METHOD Init : ITcoTaskStatus
VAR_INPUT
END_VAR
_closeTask.Restore();
Init := _closeTask.Invoke();
END_METHOD

PROPERTY InitTask : TcoCore.ITcoTask
GET
InitTask := _InitTask;
END_GET
END_PROPERTY

METHOD Open : ITcoTaskStatus
VAR_INPUT
END_VAR
_openTask.Restore();
Open := _openTask.Invoke();
END_METHOD

PROPERTY OpenTask : TcoCore.ITcoTask
GET
OpenTask := _OpenTask;
END_GET
END_PROPERTY

{warning 'Methodenimplementierung hinzufügen'}
METHOD Restore : TcoCore.ITcoRestorable
END_METHOD

{warning 'Methodenimplementierung hinzufügen'}
(*~
	<docu>
		<summary>
		    Custom service (manual, maintenance) logic.
			This method must be implemented in derived class.
		</summary>			
	</docu>	
~*)
METHOD PROTECTED ServiceMode
END_METHOD

PROPERTY Status : REFERENCE TO TcaSegmentDoorStatus
GET
Status REF= _status;
END_GET
END_PROPERTY

END_FUNCTION_BLOCK

// ---- Program/Handling/Dialogs/Handling_TeachRack_DlgContent.TcPOU
FUNCTION_BLOCK Handling_TeachRack_DlgContent EXTENDS TcoCore.TcoInputDialogContentContainer
VAR
	{attribute addProperty Name "<#Recipe#>"}
	Recipe:STRING;
	{attribute addProperty Name "<#Qantity#>"}
	RequiredQuantity:INT;
	{attribute addProperty Name "<#Timeout#>"}
	Timeout:DATE_AND_TIME;
	{attribute addProperty Name "<#Exclude#>"}
	Exclude:BOOL;
END_VAR

PROPERTY Context : TcoCore.ITcoContext
GET
END_GET
END_PROPERTY

PROPERTY Identity : ULINT
GET
END_GET
END_PROPERTY

END_FUNCTION_BLOCK

// ---- Template/Component_Cylinder/Base/CylinderBase.TcPOU
FUNCTION_BLOCK ABSTRACT CylinderBase EXTENDS TcoCore.TcoComponent IMPLEMENTS ICylinder
VAR_INPUT
	(*~
		<docu>
			<summary>
				Home position sensor.
			</summary>	
		</docu>
	~*)
	{attribute addProperty Name "<#Home position sensor#>"}
	inAtHomePos : BOOL;
	(*~
		<docu>
			<summary>
				Working position sensor.
			</summary>	
		</docu>
	~*)
	{attribute addProperty Name "<#Work position sensor#>"}
	inAtWorkPos : BOOL;
END_VAR
VAR_OUTPUT
	(*~
		<docu>
			<summary>
				Move to working home position signal.
			</summary>	
		</docu>
	~*)
	{attribute addProperty Name "<#Move to home position actuator#>"}
	outToHomePos : BOOL;
	(*~
		<docu>
			<summary>
				Move to working posistion signal.
			</summary>	
		</docu>
	~*)
	{attribute addProperty Name "<#Move to work position actuator#>"}
	outToWorkPos : BOOL;
END_VAR

(*~
	<docu>
		<summary>
			Gets whether the piston is in home position. 		
		</summary>			
	</docu>	
~*)
PROPERTY AtHome : bool
GET
AtHome := THIS^.inAtHomePos;
END_GET
END_PROPERTY

(*~
	<docu>
		<summary>
			Gets whether the piston is in work position. 		
		</summary>			
	</docu>	
~*)
PROPERTY AtWork : bool
GET
AtWork := inAtWorkPos;
END_GET
END_PROPERTY

METHOD FB_init : BOOL
VAR_INPUT
	bInitRetains : BOOL; // if TRUE, the retain variables are initialized (warm start / cold start)
	bInCopyCode : BOOL;  // if TRUE, the instance afterwards gets moved into the copy code (online change)
	Parent : ITcoObject;
END_VAR
END_METHOD

(*~
	<docu>
		<summary>
			Gets the `MoveHomeTask` task that controls the moving of the cyclinder in home position.
			<remarks>			
				<note type="important">
					This is an abstract method and must be implemented in derived class.
				</note>
			</remarks>	 		
		</summary>			
	</docu>	
~*)
PROPERTY PUBLIC ABSTRACT MoveHomeTask : TcoCore.ITcoTask
GET
END_GET
END_PROPERTY

(*~
	<docu>
		<summary>
			Starts movement into home position. 		
		</summary>			
	</docu>	
~*)
METHOD MoveToHome : TcoCore.ITcoTaskStatus
MoveToHome := MoveHomeTask.Invoke();
END_METHOD

(*~
	<docu>
		<summary>
			Starts movement into work position. 		
		</summary>			
	</docu>	
~*)
METHOD MoveToWork :TcoCore.ITcoTaskStatus
MoveToWork := MoveWorkTask.Invoke();
END_METHOD

(*~
	<docu>
		<summary>
			Gets the `MoveWorkTask` task that controls the moving of the cyclinder into work position.
			<remarks>			
				<note type="important">
					This is an abstract method and must be implemented in derived class.
				</note>
			</remarks>	 		
		</summary>			
	</docu>	
~*)
PROPERTY PUBLIC ABSTRACT MoveWorkTask : TcoCore.ITcoTask
GET
END_GET
END_PROPERTY

(*~
	<docu>
		<summary>
			Restore all tasks of this instance into initial state.		 		 		
		</summary>			
	</docu>	
~*)
METHOD  Restore : ITcoRestorable
MoveHomeTask.Restore();
MoveWorkTask.Restore();
StopTask.Restore();
END_METHOD

METHOD PROTECTED  ServiceMode
END_METHOD

(*~
	<docu>
		<summary>
			Stops cyclinder movement.
		 	<remarks>			
				<note type="important">
					This method switched off the signals for the movement of the piston in both direction.
					However depending on the pnemumatics configuration the movement may contintue if designed in that way.
					THIS IS NOT A SAFETY FUCTION!
				</note>
			</remarks>	 		
		</summary>			
	</docu>	
~*)
METHOD Stop : TcoCore.ITcoTaskStatus
Stop := StopTask.Invoke();
END_METHOD

(*~
	<docu>
		<summary>
			Gets the `StopTask` task that controls the stopping cyclinder movement.
			<remarks>			
				<note type="important">
					This is an abstract method and must be implemented in derived class.
				</note>
			</remarks>	 		
		</summary>			
	</docu>	
~*)
PROPERTY PUBLIC ABSTRACT StopTask : TcoCore.ITcoTask
GET
END_GET
END_PROPERTY

END_FUNCTION_BLOCK

// ---- Template/Component_Cylinder/Base/TcoDoubleCylinderBase.TcPOU
FUNCTION_BLOCK ABSTRACT TcoDoubleCylinderBase EXTENDS TcoCore.TcoComponent IMPLEMENTS ITcoCylinder
VAR_IN_OUT
	(*~
		<docu>
			<summary>
				Home position sensor 1.
			</summary>	
		</docu>
	~*)
	{attribute addProperty Name "<#Home position sensor#> - 1"}
	inoAtHomePos1 : BOOL;
		(*~
		<docu>
			<summary>
				Home position sensor 2.
			</summary>	
		</docu>
	~*)
	{attribute addProperty Name "<#Home position sensor#> - 2"}
	inoAtHomePos2 : BOOL;
		(*~
		<docu>
			<summary>
				Working position sensor 1.
			</summary>	
		</docu>
	~*)
	{attribute addProperty Name "<#Work position sensor#> - 1"}
	inoAtWorkPos1 : BOOL;
	(*~
		<docu>
			<summary>
				Working position sensor 1.
			</summary>	
		</docu>
	~*)
	{attribute addProperty Name "<#Work position sensor#> - 2"}
	inoAtWorkPos2 : BOOL;
END_VAR
VAR_IN_OUT
	(*~
		<docu>
			<summary>
				Move to working home position signal.
			</summary>	
		</docu>
	~*)
	{attribute addProperty Name "<#Move to home position actuator#>"}
	inoToHomePos : BOOL;
	(*~
		<docu>
			<summary>
				Move to working posistion signal.
			</summary>	
		</docu>
	~*)
	{attribute addProperty Name "<#Move to work position actuator#>"}
	inoToWorkPos : BOOL;
END_VAR
VAR
	(*~
		<docu>
			<summary>
				Home position sensor.
			</summary>	
		</docu>
	~*)
	{attribute addProperty Name "<#Home position sensor#>"}
	_atHomePos : BOOL;
	(*~
		<docu>
			<summary>
				Working position sensor.
			</summary>	
		</docu>
	~*)
	{attribute addProperty Name "<#Work position sensor#>"}
	_atWorkPos : BOOL;
	(*~
		<docu>
			<summary>
				Move to working home position signal.
			</summary>	
		</docu>
	~*)
	{attribute addProperty Name "<#Move to home position actuator#>"}
	_toHomePos : BOOL;
	(*~
		<docu>
			<summary>
				Move to working posistion signal.
			</summary>	
		</docu>
	~*)
	{attribute addProperty Name "<#Move to work position actuator#>"}
	_toWorkPos : BOOL;
END_VAR

VAR
	{attribute addProperty Name "<#Home sensor signal 1#>"}
	_atHomePos1SignalInfo : TcoCore.TcoSignalInfo;
	{attribute addProperty Name "<#Home sensor signal 2#>"}
	_atHomePos2SignalInfo : TcoCore.TcoSignalInfo;
	{attribute addProperty Name "<#Work sensor signal 1#>"}
    _atWorkPos1SignalInfo : TcoCore.TcoSignalInfo;
	{attribute addProperty Name "<#Work sensor signal 2#>"}
    _atWorkPos2SignalInfo : TcoCore.TcoSignalInfo;
	{attribute addProperty Name "<#Move to home position signal#>"}
    _toHomePosSignalInfo : TcoCore.TcoSignalInfo;
	{attribute addProperty Name "<#Move to work position signal#>"}
    _toWorkPosSignalInfo : TcoCore.TcoSignalInfo;
END_VAR

IF(__ISVALIDREF(inoAtHomePos1) AND __ISVALIDREF(inoAtHomePos2)) THEN _atHomePos := inoAtHomePos1 AND inoAtHomePos2; _atHomePos1SignalInfo.GetSignalInfo(SIZEOF(inoAtHomePos1), ADR(inoAtHomePos1));_atHomePos2SignalInfo.GetSignalInfo(SIZEOF(inoAtHomePos2), ADR(inoAtHomePos2)); END_IF;
IF(__ISVALIDREF(inoAtWorkPos1) AND __ISVALIDREF(inoAtWorkPos2)) THEN _atWorkPos := inoAtWorkPos1 AND inoAtWorkPos2; _atWorkPos1SignalInfo.GetSignalInfo(SIZEOF(inoAtWorkPos1), ADR(inoAtWorkPos1));_atWorkPos2SignalInfo.GetSignalInfo(SIZEOF(inoAtWorkPos2), ADR(inoAtWorkPos2)); END_IF;
IF(__ISVALIDREF(inoToHomePos)) THEN inoToHomePos := _toHomePos; _toHomePosSignalInfo.GetSignalInfo(SIZEOF(inoToHomePos), ADR(inoToHomePos)); END_IF;
IF(__ISVALIDREF(inoToWorkPos)) THEN inoToWorkPos := _toWorkPos; _toWorkPosSignalInfo.GetSignalInfo(SIZEOF(inoToWorkPos), ADR(inoToWorkPos)); END_IF;

(*~
	<docu>
		<summary>
			Gets whether the piston is in home position. 		
		</summary>			
	</docu>	
~*)
PROPERTY AtHome : bool
GET
AtHome := THIS^._atHomePos;
END_GET
END_PROPERTY

(*~
	<docu>
		<summary>
			Gets whether the piston is in work position. 		
		</summary>			
	</docu>	
~*)
PROPERTY AtWork : bool
GET
AtWork := _atWorkPos;
END_GET
END_PROPERTY

METHOD FB_init : BOOL
VAR_INPUT
	bInitRetains : BOOL; // if TRUE, the retain variables are initialized (warm start / cold start)
	bInCopyCode : BOOL;  // if TRUE, the instance afterwards gets moved into the copy code (online change)
	ParentObject : ITcoObject;	
END_VAR
END_METHOD

(*~
	<docu>
		<summary>
			Gets the `MoveHomeTask` task that controls the moving of the cyclinder in home position.
			<remarks>			
				<note type="important">
					This is an abstract method and must be implemented in derived class.
				</note>
			</remarks>	 		
		</summary>			
	</docu>	
~*)
PROPERTY PUBLIC ABSTRACT MoveHomeTask : TcoCore.ITcoTask
GET
END_GET
END_PROPERTY

(*~
	<docu>
		<summary>
			Starts movement into home position. 		
		</summary>			
	</docu>	
~*)
METHOD MoveToHome : TcoCore.ITcoTaskStatus
IF(MoveHomeTask <> 0) THEN 
	MoveToHome := MoveHomeTask.Invoke();
END_IF;
END_METHOD

(*~
	<docu>
		<summary>
			Starts movement into work position. 		
		</summary>			
	</docu>	
~*)
METHOD MoveToWork :TcoCore.ITcoTaskStatus
IF(MoveWorkTask <> 0) THEN
	MoveToWork := MoveWorkTask.Invoke();
END_IF;
END_METHOD

(*~
	<docu>
		<summary>
			Gets the `MoveWorkTask` task that controls the moving of the cyclinder into work position.
			<remarks>			
				<note type="important">
					This is an abstract method and must be implemented in derived class.
				</note>
			</remarks>	 		
		</summary>			
	</docu>	
~*)
PROPERTY PUBLIC ABSTRACT MoveWorkTask : TcoCore.ITcoTask
GET
END_GET
END_PROPERTY

(*~
	<docu>
		<summary>
			Restore all tasks of this instance into initial state.		 		 		
		</summary>			
	</docu>	
~*)
METHOD  Restore : ITcoRestorable
IF(MoveHomeTask <> 0) THEN MoveHomeTask.Restore(); END_IF;
IF(MoveWorkTask <> 0) THEN MoveWorkTask.Restore(); END_IF;
IF(StopTask <> 0) THEN StopTask.Restore(); END_IF;
END_METHOD

METHOD PROTECTED  ServiceMode
END_METHOD

(*~
	<docu>
		<summary>
			Stops cyclinder movement.
		 	<remarks>			
				<note type="important">
					This method switched off the signals for the movement of the piston in both direction.
					However depending on the pnemumatics configuration the movement may contintue if designed in that way.
					THIS IS NOT A SAFETY FUCTION!
				</note>
			</remarks>	 		
		</summary>			
	</docu>	
~*)
METHOD Stop : TcoCore.ITcoTaskStatus
IF(StopTask <> 0) THEN
	Stop := StopTask.Invoke();
END_IF;
END_METHOD

(*~
	<docu>
		<summary>
			Gets the `StopTask` task that controls the stopping cyclinder movement.
			<remarks>			
				<note type="important">
					This is an abstract method and must be implemented in derived class.
				</note>
			</remarks>	 		
		</summary>			
	</docu>	
~*)
PROPERTY PUBLIC ABSTRACT StopTask : TcoCore.ITcoTask
GET
END_GET
END_PROPERTY

END_FUNCTION_BLOCK

// ---- Template/Component_Cylinder/Tasks/CylinderMoveTask.TcPOU
FUNCTION_BLOCK CylinderMoveTask EXTENDS TcoCore.TcoTask
VAR_INPUT
	PositionSensor		   : BOOL;
	MaxTimeToReachPosition : TIME := T#10S;
	PositionName		   : STRING(25);
END_VAR
VAR_IN_OUT
	MoveToPositionSignal : BOOL;
	InverseSignal		 : BOOL;	
END_VAR

VAR
	_stringBuilder : TcoCore.StringBuilder;
END_VAR

IF (THIS^.Execute()) THEN
	IF(THIS^.ElapsedTime > MaxTimeToReachPosition) THEN THIS^.Messenger.Warning(_stringBuilder.Clear().Append(PositionName).Append(' sensor not reached yet.').ToString()); END_IF;
	InverseSignal		 := FALSE;
	MoveToPositionSignal := TRUE;
	THIS^DoneWhen(PositionSensor);
END_IF

METHOD PUBLIC FB_init : BOOL
VAR_INPUT
	bInitRetains : BOOL; // if TRUE, the retain variables are initialized (warm start / cold start)
	bInCopyCode : BOOL;  // if TRUE, the instance afterwards gets moved into the copy code (online change)
	Parent : ITcoObject;
END_VAR
END_METHOD

(*~
	<docu>
		<summary>
			Executes when task is aborted.
		</summary>			
	</docu>	
~*)
METHOD PROTECTED OnAbort
MoveToPositionSignal := FALSE;
END_METHOD

END_FUNCTION_BLOCK

// ---- Template/Component_Cylinder/TcoCylinder.TcPOU
{attribute addProperty _moveHomeDefaultName "<#MOVE HOME#>"}
{attribute addProperty _moveWorkDefaultName "<#MOVE TO WORK#>"}
{attribute addProperty _stopDefaultName "<#STOP#>"}
FUNCTION_BLOCK TcoCylinder EXTENDS TcoCylinderBase
VAR
    {attribute addProperty Name "|[[1]Attribute_moveHomeDefaultName]|"}
    _moveHomeDefault : TcoCylinderMoveTask(THIS^);
    {attribute addProperty Name "|[[1]Attribute_moveWorkDefaultName]|"}
    _moveWorkDefault : TcoCylinderMoveTask(THIS^);
    {attribute addProperty Name "|[[1]Attribute_stopDefaultName]|"}
    _stopDefault : TcoCore.TcoTask(THIS^);
	increment: INT;
END_VAR
VAR
    _config : TcoCylinderConfig;
	_status : TcoCylinderStatus;
	_refillTimer:TON;	
END_VAR

SUPER^(inoAtHomePos := inoAtHomePos, inoAtWorkPos := inoAtWorkPos, inoToHomePos := inoToHomePos, inoToWorkPos := inoToWorkPos);
	
IF(_atHomePos AND _atWorkPos) THEN Messenger.Error('<#Home and work position sensors are both active. Check the position of sensors!#>'); END_IF;

// Disables mutualy exclusive actions
_moveWorkDefault.Enabled := TRUE;// NOT _moveHomeDefault.Busy;


_moveHomeDefault(PositionSensor := _atHomePos AND NOT _atWorkPos,
    MoveToPositionSignal := _toHomePos,
    InverseSignal := _toWorkPos,
	TimeToRefill:=_config.TimeToRefill,
    MaxTimeToReachPosition := _config.TimeToReachHomePosition,
    PositionName := '<#Home#>');

IF _moveHomeDefault.Execute() THEN
	_moveWorkDefault.Restore();
END_IF
	
// Disables mutualy exclusive actions		
_moveHomeDefault.Enabled := TRUE;//NOT _moveWorkDefault.Busy;
	
_moveWorkDefault(PositionSensor := _atWorkPos AND NOT _atHomePos,
    MoveToPositionSignal := _toWorkPos,
    InverseSignal := _toHomePos,
	TimeToRefill:=_config.TimeToRefill,
    MaxTimeToReachPosition := _config.TimeToReachWorkPosition,
    PositionName := '<#Work#>');
	
IF _moveWorkDefault.Execute() THEN
	_moveHomeDefault.Restore();
END_IF

IF (_stopDefault.Execute()) THEN
	_toHomePos := FALSE;
	_toWorkPos := FALSE;
    _moveHomeDefault.Abort();
    _moveWorkDefault.Abort();
    _stopDefault.Abort();
    _moveHomeDefault.Restore();
    _moveWorkDefault.Restore();
    _stopDefault.Restore();
    _stopDefault.DoneWhen(TRUE);
END_IF

// For further discussion about Status
IF(_moveHomeDefault.Busy) THEN
	_status.ActionDescription := 'Moving to home position';
ELSIF(_moveWorkDefault.Busy) THEN
	_status.ActionDescription := 'Moving to work position';
ELSIF(_stopDefault.Busy) THEN
	_status.ActionDescription := 'Stopping pressure';
ELSE	
	_status.ActionDescription := 'Idle';
END_IF

SUPER^(inoAtHomePos := inoAtHomePos, inoAtWorkPos := inoAtWorkPos, inoToHomePos := inoToHomePos, inoToWorkPos := inoToWorkPos);

(*~
	<docu>
		<summary>
			Aborts the movement to home position when the condition is 'true'.
		</summary>
		<remarks>			
				<note type="warning">
					The call of this method will be effective only when called AFTER the initialization of the instance of given TcoCylinder.
				</note>
		</remarks>	
	</docu>
~*)
METHOD AbortMoveHome : BOOL
VAR_IN_OUT
	(*~
	<docu>
		<summary>
			Condition to abort the movement of the cylinder.
		</summary>	
	</docu>
	~*)
	inoDisableCondition : BOOL;
END_VAR
VAR
	_signalInfo : TcoSignalInfo;
END_VAR
IF (_toHomePos OR _moveHomeDefault.Busy) AND inoDisableCondition THEN
	_signalInfo.GetSignalInfo(SIZEOF(inoDisableCondition), ADR(inoDisableCondition));
	Messenger.Build().Append('<#Movement aborted due to#> : ').Append(_signalInfo.SymbolPath).As().AsError().Pin();
	_toHomePos := FALSE;
	IF(__ISVALIDREF(THIS^.inoToHomePos)) THEN THIS^.inoToHomePos := FALSE; END_IF;
	_moveHomeDefault.Abort();
END_IF
END_METHOD

(*~
	<docu>
		<summary>
			Aborts the movement to work position when the condition is 'true'.
		</summary>
		<remarks>			
				<note type="warning">
					The call of this method will be effective only when called AFTER the initialization of the instance of given TcoCylinder.
				</note>
		</remarks>	
	</docu>
~*)
METHOD AbortMoveWork : BOOL
VAR_IN_OUT
	(*~
		<docu>
			<summary>
				Condition to abort the movement of the cylinder.
			</summary>	
		</docu>
	~*)
	inoDisableCondition : BOOL;
END_VAR
VAR
	_signalInfo : TcoSignalInfo;
END_VAR
IF (_toWorkPos OR _moveWorkDefault.Busy) AND inoDisableCondition THEN
	_signalInfo.GetSignalInfo(SIZEOF(inoDisableCondition), ADR(inoDisableCondition));
	Messenger.Build().Append('<#Movement aborted due to#> : ').Append(_signalInfo.SymbolPath).As().AsError().Pin();
	_toWorkPos := FALSE;
	IF(__ISVALIDREF(THIS^.inoToWorkPos)) THEN THIS^.inoToWorkPos := FALSE; END_IF;
	_moveWorkDefault.Abort();
END_IF
END_METHOD

(*~
	<docu>
		<summary>
			Gets the configuration of the cylinder. 					
		</summary>			
	</docu>	
~*)
PROPERTY Config : REFERENCE TO TcoCylinderConfig
GET
Config REF= _config;
END_GET
END_PROPERTY

(*~
	<docu>
		<summary>
			Gets the `MoveHomeTask` task that controls the moving of the cyclinder in home position. 		
		</summary>			
	</docu>	
~*)
PROPERTY MoveHomeTask : TcoCore.ITcoTask
GET
MoveHomeTask := _moveHomeDefault;
END_GET
END_PROPERTY

(*~
	<docu>
		<summary>
			Gets the `MoveWorkTask` task that controls the moving of the cyclinder into work position. 		
		</summary>			
	</docu>	
~*)
PROPERTY MoveWorkTask : TcoCore.ITcoTask
GET
MoveWorkTask := _moveWorkDefault;
END_GET
END_PROPERTY

(*~
	<docu>
		<summary>
			Refill cylinder after booth outputs are off .
		</summary>
		<remarks>			
				<note type="warning">
					The call of this method will be effective only when called AFTER the initialization of the instance of given TcoCylinder and methods like AbortMoveHone,SuspendMoveHom...
				</note>
		</remarks>	
	</docu>
~*)
METHOD Refill : BOOL
VAR_INPUT
	(*~
	<docu>
		<summary>
			Time of refill cylinder after aborting or suspending
		</summary>	
	</docu>
	~*)
	inRefillTime:TIME;
END_VAR

_refillTimer(In:=inoToHomePos XOR  inoToWorkPos ,Pt:=T#49D);

_config.TimeToRefill:=inRefillTime;

IF  _refillTimer.ET>T#0MS
	AND _refillTimer.ET<_config.TimeToRefill  
	AND _config.TimeToRefill<>T#0S THEN
	_toHomePos	 := TRUE;
	_toWorkPos	 := TRUE;	
END_IF;

	
SUPER^(inoAtHomePos := inoAtHomePos, inoAtWorkPos := inoAtWorkPos, inoToHomePos := inoToHomePos, inoToWorkPos := inoToWorkPos);
END_METHOD

PROPERTY Status : REFERENCE TO TcoCylinderStatus
GET
Status REF= _status;
END_GET
END_PROPERTY

(*~
	<docu>
		<summary>
			Gets the `StopTask` task that controls the stopping of the cyclinder. 		
		</summary>			
	</docu>	
~*)
PROPERTY StopTask : TcoCore.ITcoTask
GET
StopTask := _stopDefault;
END_GET
END_PROPERTY

(*~
	<docu>
		<summary>
			Suspend the movement to home position when the condition is 'true'. Task is still busy
		</summary>
		<remarks>			
				<note type="warning">
					The call of this method will be effective only when called AFTER the initialization of the instance of given TcoCylinder.
				</note>
		</remarks>	
	</docu>
~*)
METHOD SuspendMoveHome : BOOL
VAR_IN_OUT
	(*~
	<docu>
		<summary>
			Condition to abort the movement of the cylinder.
		</summary>	
	</docu>
	~*)
	inoDisableCondition : BOOL;
END_VAR
VAR
	_signalInfo : TcoSignalInfo;
END_VAR
IF (_toHomePos OR _moveHomeDefault.Busy) AND inoDisableCondition THEN
	_signalInfo.GetSignalInfo(SIZEOF(inoDisableCondition), ADR(inoDisableCondition));
	Messenger.Warning(CONCAT('<#Movement suspended due to#> : ' , _signalInfo.SymbolPath));
	_toHomePos := FALSE;
	IF(__ISVALIDREF(THIS^.inoToHomePos)) THEN THIS^.inoToHomePos := FALSE; END_IF;
	
END_IF
END_METHOD

METHOD SuspendMoveHomeExpression : BOOL
VAR_INPUT
		inDisableCondition : BOOL;
		inMessage:STRING;
END_VAR
IF (_toHomePos OR _moveHomeDefault.Busy) AND inDisableCondition THEN
	Messenger.Warning(CONCAT('<#Movement suspended due to#> : ' , inMessage));
	_toHomePos := FALSE;
	IF(__ISVALIDREF(THIS^.inoToHomePos)) THEN THIS^.inoToHomePos := FALSE; END_IF;
	
END_IF;
END_METHOD

(*~
	<docu>
		<summary>
			Suspend the movement to home position when the condition is NOT 'true'. Task is still busy
		</summary>
		<remarks>			
				<note type="warning">
					The call of this method will be effective only when called AFTER the initialization of the instance of given TcoCylinder.
				</note>
		</remarks>	
	</docu>
~*)
METHOD SuspendMoveHomeInverted : BOOL
VAR_IN_OUT
	(*~
	<docu>
		<summary>
			Condition to abort the movement of the cylinder.
		</summary>	
	</docu>
	~*)
	inoDisableCondition : BOOL;
END_VAR
VAR
	_signalInfo : TcoSignalInfo;
END_VAR
IF (_toHomePos OR _moveHomeDefault.Busy) AND not inoDisableCondition THEN
	_signalInfo.GetSignalInfo(SIZEOF(inoDisableCondition), ADR(inoDisableCondition));
	Messenger.Warning(CONCAT('<#Movement suspended due to NOT#> : ' , _signalInfo.SymbolPath));
	_toHomePos := FALSE;
	IF(__ISVALIDREF(THIS^.inoToHomePos)) THEN THIS^.inoToHomePos := FALSE; END_IF;
	
END_IF
END_METHOD

(*~
	<docu>
		<summary>
			Suspend the movement to work position when the condition is 'true'. Task is still bussy
		</summary>
		<remarks>			
				<note type="warning">
					The call of this method will be effective only when called AFTER the initialization of the instance of given TcoCylinder.
				</note>
		</remarks>	
	</docu>
~*)
METHOD SuspendMoveWork : BOOL
VAR_IN_OUT
	(*~
		<docu>
			<summary>
				Condition to abort the movement of the cylinder.
			</summary>	
		</docu>
	~*)
	inoDisableCondition : BOOL;
END_VAR
VAR
	_signalInfo : TcoSignalInfo;
END_VAR
IF (_toWorkPos OR _moveWorkDefault.Busy) AND inoDisableCondition THEN
	_signalInfo.GetSignalInfo(SIZEOF(inoDisableCondition), ADR(inoDisableCondition));
	Messenger.Warning(CONCAT('<#Movement suspended due to#> : ' , _signalInfo.SymbolPath));
	_toWorkPos := FALSE;
	IF(__ISVALIDREF(THIS^.inoToWorkPos)) THEN THIS^.inoToWorkPos := FALSE; END_IF;

END_IF
END_METHOD

METHOD SuspendMoveWorkExpression : BOOL
VAR_INPUT
		inDisableCondition : BOOL;
		inMessage:STRING;
END_VAR
IF (_toWorkPos OR _moveWorkDefault.Busy) AND inDisableCondition THEN
	Messenger.Warning(CONCAT('<#Movement suspended due to#> : ' , inMessage));
	_toWorkPos := FALSE;
	IF(__ISVALIDREF(THIS^.inoToWorkPos)) THEN THIS^.inoToWorkPos := FALSE; END_IF;
	
END_IF
END_METHOD

(*~
	<docu>
		<summary>
			Suspend the movement to work position when the condition is NOT 'true'. Task is still busy
		</summary>
		<remarks>			
				<note type="warning">
					The call of this method will be effective only when called AFTER the initialization of the instance of given TcoCylinder.
				</note>
		</remarks>	
	</docu>
~*)
METHOD SuspendMoveWorkInverted : BOOL
VAR_IN_OUT
	(*~
		<docu>
			<summary>
				Condition to abort the movement of the cylinder.
			</summary>	
		</docu>
	~*)
	inoDisableCondition : BOOL;
END_VAR
VAR
	_signalInfo : TcoSignalInfo;
END_VAR
IF (_toWorkPos OR _moveWorkDefault.Busy) AND not inoDisableCondition THEN
	_signalInfo.GetSignalInfo(SIZEOF(inoDisableCondition), ADR(inoDisableCondition));
	Messenger.Warning(CONCAT('<#Movement suspended due to NOT#> : ' , _signalInfo.SymbolPath));
	_toWorkPos := FALSE;
	IF(__ISVALIDREF(THIS^.inoToWorkPos)) THEN THIS^.inoToWorkPos := FALSE; END_IF;

END_IF
END_METHOD

END_FUNCTION_BLOCK

// ---- Template/Component_Cylinder/TcoDoubleCylinder.TcPOU
{attribute addProperty _moveHomeDefaultName "<#MOVE HOME#>"}
{attribute addProperty _moveWorkDefaultName "<#MOVE TO WORK#>"}
{attribute addProperty _stopDefaultName "<#STOP#>"}
FUNCTION_BLOCK TcoDoubleCylinder EXTENDS TcoDoubleCylinderBase
VAR
    {attribute addProperty Name "|[[1]Attribute_moveHomeDefaultName]|"}
    _moveHomeDefault : TcoCylinderMoveTask(THIS^);
    {attribute addProperty Name "|[[1]Attribute_moveWorkDefaultName]|"}
    _moveWorkDefault : TcoCylinderMoveTask(THIS^);
    {attribute addProperty Name "|[[1]Attribute_stopDefaultName]|"}
    _stopDefault : TcoCore.TcoTask(THIS^);
	increment: INT;

END_VAR
VAR
    _config : TcoCylinderConfig;
	_status : TcoCylinderStatus;
	_refillTimer:TON;	
END_VAR

SUPER^(inoAtHomePos1 := inoAtHomePos1,inoAtHomePos2 := inoAtHomePos2, inoAtWorkPos1 := inoAtWorkPos1,inoAtWorkPos2 := inoAtWorkPos2, inoToHomePos := inoToHomePos, inoToWorkPos := inoToWorkPos);
	
IF(_atHomePos AND _atWorkPos) THEN Messenger.Error('<#Home and work position sensors are both active. Check the position of sensors!#>'); END_IF;

// Disables mutualy exclusive actions
_moveWorkDefault.Enabled :=TRUE;// NOT _moveHomeDefault.Busy;

_moveHomeDefault(PositionSensor := _atHomePos AND NOT _atWorkPos,
    MoveToPositionSignal := _toHomePos,
    InverseSignal := _toWorkPos,
	TimeToRefill:=_config.TimeToRefill,
    MaxTimeToReachPosition := _config.TimeToReachHomePosition,
    PositionName := '<#Home#>');
IF _moveHomeDefault.Execute() THEN
	_moveWorkDefault.Restore();
END_IF

// Disables mutualy exclusive actions		
_moveHomeDefault.Enabled :=true;// NOT _moveWorkDefault.Busy;
	
_moveWorkDefault(PositionSensor := _atWorkPos AND NOT _atHomePos,
    MoveToPositionSignal := _toWorkPos,
    InverseSignal := _toHomePos,
	TimeToRefill:=_config.TimeToRefill,
    MaxTimeToReachPosition := _config.TimeToReachWorkPosition,
    PositionName := '<#Work#>');

IF _moveWorkDefault.Execute() THEN
	_moveHomeDefault.Restore();
END_IF


IF (_stopDefault.Execute()) THEN
	_toHomePos := FALSE;
	_toWorkPos := FALSE;
    _moveHomeDefault.Abort();
    _moveWorkDefault.Abort();
    _stopDefault.Abort();
    _moveHomeDefault.Restore();
    _moveWorkDefault.Restore();
    _stopDefault.Restore();
    _stopDefault.DoneWhen(TRUE);
END_IF

// For further discussion about Status
IF(_moveHomeDefault.Busy) THEN
	_status.ActionDescription := 'Moving to home position';
ELSIF(_moveWorkDefault.Busy) THEN
	_status.ActionDescription := 'Moving to work position';
ELSIF(_stopDefault.Busy) THEN
	_status.ActionDescription := 'Stopping pressure';
ELSE	
	_status.ActionDescription := 'Idle';
END_IF

SUPER^(inoAtHomePos1 := inoAtHomePos1,inoAtHomePos2 := inoAtHomePos2, inoAtWorkPos1 := inoAtWorkPos1,inoAtWorkPos2 := inoAtWorkPos2, inoToHomePos := inoToHomePos, inoToWorkPos := inoToWorkPos);

(*~
	<docu>
		<summary>
			Aborts the movement to home position when the condition is 'true'.
		</summary>
		<remarks>			
				<note type="warning">
					The call of this method will be effective only when called AFTER the initialization of the instance of given TcoCylinder.
				</note>
		</remarks>	
	</docu>
~*)
METHOD AbortMoveHome : BOOL
VAR_IN_OUT
	(*~
	<docu>
		<summary>
			Condition to abort the movement of the cylinder.
		</summary>	
	</docu>
	~*)
	inoDisableCondition : BOOL;
END_VAR
VAR
	_signalInfo : TcoSignalInfo;
END_VAR
IF (_toHomePos OR _moveHomeDefault.Busy) AND inoDisableCondition THEN
	_signalInfo.GetSignalInfo(SIZEOF(inoDisableCondition), ADR(inoDisableCondition));
	Messenger.Build().Append('<#Movement aborted due to#> : ').Append(_signalInfo.SymbolPath).As().AsError().Pin();
	_toHomePos := FALSE;
	IF(__ISVALIDREF(THIS^.inoToHomePos)) THEN THIS^.inoToHomePos := FALSE; END_IF;
	_moveHomeDefault.Abort();
END_IF
END_METHOD

(*~
	<docu>
		<summary>
			Aborts the movement to work position when the condition is 'true'.
		</summary>
		<remarks>			
				<note type="warning">
					The call of this method will be effective only when called AFTER the initialization of the instance of given TcoCylinder.
				</note>
		</remarks>	
	</docu>
~*)
METHOD AbortMoveWork : BOOL
VAR_IN_OUT
	(*~
		<docu>
			<summary>
				Condition to abort the movement of the cylinder.
			</summary>	
		</docu>
	~*)
	inoDisableCondition : BOOL;
END_VAR
VAR
	_signalInfo : TcoSignalInfo;
END_VAR
IF (_toWorkPos OR _moveWorkDefault.Busy) AND inoDisableCondition THEN
	_signalInfo.GetSignalInfo(SIZEOF(inoDisableCondition), ADR(inoDisableCondition));
	Messenger.Build().Append('<#Movement aborted due to#> : ').Append(_signalInfo.SymbolPath).As().AsError().Pin();
	_toWorkPos := FALSE;
	IF(__ISVALIDREF(THIS^.inoToWorkPos)) THEN THIS^.inoToWorkPos := FALSE; END_IF;
	_moveWorkDefault.Abort();
END_IF
END_METHOD

(*~
	<docu>
		<summary>
			Gets the configuration of the cylinder. 					
		</summary>			
	</docu>	
~*)
PROPERTY Config : REFERENCE TO TcoCylinderConfig
GET
Config REF= _config;
END_GET
END_PROPERTY

(*~
	<docu>
		<summary>
			Gets the `MoveHomeTask` task that controls the moving of the cyclinder in home position. 		
		</summary>			
	</docu>	
~*)
PROPERTY MoveHomeTask : TcoCore.ITcoTask
GET
MoveHomeTask := _moveHomeDefault;
END_GET
END_PROPERTY

(*~
	<docu>
		<summary>
			Gets the `MoveWorkTask` task that controls the moving of the cyclinder into work position. 		
		</summary>			
	</docu>	
~*)
PROPERTY MoveWorkTask : TcoCore.ITcoTask
GET
MoveWorkTask := _moveWorkDefault;
END_GET
END_PROPERTY

(*~
	<docu>
		<summary>
			Refill cylinder after booth outputs are off .
		</summary>
		<remarks>			
				<note type="warning">
					The call of this method will be effective only when called AFTER the initialization of the instance of given TcoCylinder and methods like AbortMoveHone,SuspendMoveHom...
				</note>
		</remarks>	
	</docu>
~*)
METHOD Refill : BOOL
VAR_INPUT
	(*~
	<docu>
		<summary>
			Time of refill cylinder after aborting or suspending
		</summary>	
	</docu>
	~*)
	inRefillTime:TIME;
END_VAR

_refillTimer(In:=inoToHomePos XOR  inoToWorkPos ,Pt:=T#49D);

_config.TimeToRefill:=inRefillTime;

IF  _refillTimer.ET>T#0MS
	AND _refillTimer.ET<_config.TimeToRefill  
	AND _config.TimeToRefill<>T#0S THEN
	_toHomePos	 := TRUE;
	_toWorkPos	 := TRUE;	
END_IF;

	
SUPER^(inoAtHomePos1 := inoAtHomePos1,inoAtHomePos2 := inoAtHomePos2, inoAtWorkPos1 := inoAtWorkPos1,inoAtWorkPos2 := inoAtWorkPos2, inoToHomePos := inoToHomePos, inoToWorkPos := inoToWorkPos);
END_METHOD

PROPERTY Status : REFERENCE TO TcoCylinderStatus
GET
Status REF= _status;
END_GET
END_PROPERTY

(*~
	<docu>
		<summary>
			Gets the `StopTask` task that controls the stopping of the cyclinder. 		
		</summary>			
	</docu>	
~*)
PROPERTY StopTask : TcoCore.ITcoTask
GET
StopTask := _stopDefault;
END_GET
END_PROPERTY

(*~
	<docu>
		<summary>
			Suspend the movement to home position when the condition is 'true'. Task is still busy
		</summary>
		<remarks>			
				<note type="warning">
					The call of this method will be effective only when called AFTER the initialization of the instance of given TcoCylinder.
				</note>
		</remarks>	
	</docu>
~*)
METHOD SuspendMoveHome : BOOL
VAR_IN_OUT
	(*~
	<docu>
		<summary>
			Condition to abort the movement of the cylinder.
		</summary>	
	</docu>
	~*)
	inoDisableCondition : BOOL;
END_VAR
VAR
	_signalInfo : TcoSignalInfo;
END_VAR
IF (_toHomePos OR _moveHomeDefault.Busy) AND inoDisableCondition THEN
	_signalInfo.GetSignalInfo(SIZEOF(inoDisableCondition), ADR(inoDisableCondition));
	Messenger.Warning(CONCAT('<#Movement suspended due to#> : ' , _signalInfo.SymbolPath));
	_toHomePos := FALSE;
	IF(__ISVALIDREF(THIS^.inoToHomePos)) THEN THIS^.inoToHomePos := FALSE; END_IF;
	
END_IF
END_METHOD

METHOD SuspendMoveHomeExpression : BOOL
VAR_INPUT
		inDisableCondition : BOOL;
		inMessage:STRING;
END_VAR
IF (_toHomePos OR _moveHomeDefault.Busy) AND inDisableCondition THEN
	Messenger.Warning(CONCAT('<#Movement suspended due to#> : ' , inMessage));
	_toHomePos := FALSE;
	IF(__ISVALIDREF(THIS^.inoToHomePos)) THEN THIS^.inoToHomePos := FALSE; END_IF;
	
END_IF;
END_METHOD

(*~
	<docu>
		<summary>
			Suspend the movement to home position when the condition is NOT 'true'. Task is still busy
		</summary>
		<remarks>			
				<note type="warning">
					The call of this method will be effective only when called AFTER the initialization of the instance of given TcoCylinder.
				</note>
		</remarks>	
	</docu>
~*)
METHOD SuspendMoveHomeInverted : BOOL
VAR_IN_OUT
	(*~
	<docu>
		<summary>
			Condition to abort the movement of the cylinder.
		</summary>	
	</docu>
	~*)
	inoDisableCondition : BOOL;
END_VAR
VAR
	_signalInfo : TcoSignalInfo;
END_VAR
IF (_toHomePos OR _moveHomeDefault.Busy) AND NOT inoDisableCondition THEN
	_signalInfo.GetSignalInfo(SIZEOF(inoDisableCondition), ADR(inoDisableCondition));
	Messenger.Warning(CONCAT('<#Movement suspended due to NOT#> : ' , _signalInfo.SymbolPath));
	_toHomePos := FALSE;
	IF(__ISVALIDREF(THIS^.inoToHomePos)) THEN THIS^.inoToHomePos := FALSE; END_IF;
	
END_IF
END_METHOD

(*~
	<docu>
		<summary>
			Suspend the movement to work position when the condition is 'true'. Task is still bussy
		</summary>
		<remarks>			
				<note type="warning">
					The call of this method will be effective only when called AFTER the initialization of the instance of given TcoCylinder.
				</note>
		</remarks>	
	</docu>
~*)
METHOD SuspendMoveWork : BOOL
VAR_IN_OUT
	(*~
		<docu>
			<summary>
				Condition to abort the movement of the cylinder.
			</summary>	
		</docu>
	~*)
	inoDisableCondition : BOOL;
END_VAR
VAR
	_signalInfo : TcoSignalInfo;
END_VAR
IF (_toWorkPos OR _moveWorkDefault.Busy) AND inoDisableCondition THEN
	_signalInfo.GetSignalInfo(SIZEOF(inoDisableCondition), ADR(inoDisableCondition));
	Messenger.Warning(CONCAT('<#Movement suspended due to#> : ' , _signalInfo.SymbolPath));
	_toWorkPos := FALSE;
	IF(__ISVALIDREF(THIS^.inoToWorkPos)) THEN THIS^.inoToWorkPos := FALSE; END_IF;

END_IF
END_METHOD

METHOD SuspendMoveWorkExpression : BOOL
VAR_INPUT
		inDisableCondition : BOOL;
		inMessage:STRING;
END_VAR
IF (_toWorkPos OR _moveWorkDefault.Busy) AND inDisableCondition THEN
	Messenger.Warning(CONCAT('<#Movement suspended due to#> : ' , inMessage));
	_toWorkPos := FALSE;
	IF(__ISVALIDREF(THIS^.inoToWorkPos)) THEN THIS^.inoToWorkPos := FALSE; END_IF;
	
END_IF
END_METHOD

(*~
	<docu>
		<summary>
			Suspend the movement to work position when the condition is NOT 'true'. Task is still bussy
		</summary>
		<remarks>			
				<note type="warning">
					The call of this method will be effective only when called AFTER the initialization of the instance of given TcoCylinder.
				</note>
		</remarks>	
	</docu>
~*)
METHOD SuspendMoveWorkInverted : BOOL
VAR_IN_OUT
	(*~
		<docu>
			<summary>
				Condition to abort the movement of the cylinder.
			</summary>	
		</docu>
	~*)
	inoDisableCondition : BOOL;
END_VAR
VAR
	_signalInfo : TcoSignalInfo;
END_VAR
IF (_toWorkPos OR _moveWorkDefault.Busy) AND NOT inoDisableCondition THEN
	_signalInfo.GetSignalInfo(SIZEOF(inoDisableCondition), ADR(inoDisableCondition));
	Messenger.Warning(CONCAT('<#Movement suspended due to NOT#> : ' , _signalInfo.SymbolPath));
	_toWorkPos := FALSE;
	IF(__ISVALIDREF(THIS^.inoToWorkPos)) THEN THIS^.inoToWorkPos := FALSE; END_IF;

END_IF
END_METHOD

END_FUNCTION_BLOCK

// ---- Template/RackFeeder/FB_RackFeeder.TcPOU
FUNCTION_BLOCK FB_RackFeeder EXTENDS FB_Component

VAR CONSTANT
	nTrolleyDockCount				: INT := 3;
	nStorageDockCount				: INT := 5;
END_VAR

VAR
	bSimulation						: BOOL;
	
	fbAxisTraverse					: FB_AxisDriver;
	fbAxisLift						: FB_AxisDriver;
	fbAxisTelescope					: FB_AxisDriver;	
	
	fEndposTraverse					: LREAL;
	fEndposLift						: LREAL;
	fEndposTelescope				: LREAL;
	
	fbCarrierPresent				: FB_DigitalInput;

	aTrolleyDocks					: ARRAY[0..nTrolleyDockCount] OF ST_TrolleyDock;	
	aStorageDocks					: ARRAY[0..nStorageDockCount] OF ST_StorageDock;
	
	aJobs							: ARRAY[0..127] OF ST_RackFeederJob;	
END_VAR

VAR_OUTPUT
	Carrier							: FB_WorkpieceCarrier;
END_VAR

VAR_INPUT
	cmd								: CMD_RackFeeder;
END_VAR

METHOD DropCarrier : BOOL
VAR_INPUT
END_VAR
END_METHOD

METHOD FetchCarrier : BOOL
VAR_INPUT
END_VAR
END_METHOD

METHOD FindCarrier
VAR_INPUT
END_VAR
END_METHOD

METHOD RegisterStorageDock
VAR_IN_OUT
	Storage				: FB_Storage;
END_VAR


VAR
	ni						: INT;
END_VAR
// Search if Reference is already in List
FOR ni := 0 TO nStorageDockCount DO

	IF NOT __ISVALIDREF(aTrolleyDocks[ni].refTrolley) THEN
		aStorageDocks[ni].refStorage REF= Storage;	
		EXIT;
	END_IF
	
	IF ADR(aStorageDocks[ni].refStorage) <> ADR(Storage) THEN
		CONTINUE;
	ELSE
		EXIT;
	END_IF

END_FOR
END_METHOD

METHOD RegisterTrolleyDock
VAR_IN_OUT
	Trolley				: FB_Trolley;
END_VAR

VAR
	ni						: INT;
END_VAR

// Search if Reference is already in List
FOR ni := 0 TO nTrolleyDockCount DO

	IF NOT __ISVALIDREF(aTrolleyDocks[ni].refTrolley) THEN
		aTrolleyDocks[ni].refTrolley REF= Trolley;	
		EXIT;
	END_IF
	
	IF ADR(aTrolleyDocks[ni].refTrolley) <> ADR(Trolley) THEN
		CONTINUE;
	ELSE
		EXIT;
	END_IF

END_FOR
END_METHOD

/// RunSuper component logic
{attribute 'object_name' := 'Run'}
METHOD  Run
// Component Run
fbAxisTraverse.Run();
fbAxisLift.Run();
fbAxisTelescope.Run();

fEndposTraverse := 3000;
fEndposLift := 900;
fEndposTelescope := 1800;

// Axis Run
fbAxisTraverse.Enable := TRUE;
fbAxisTraverse.EnableCtrl := TRUE;
fbAxisTraverse.EnableNeg := TRUE;
fbAxisTraverse.EnablePos := TRUE;
fbAxisTraverse.Override := 100; //TODO: Höher stellen
fbAxisTraverse.TorqueLimit := 10; //TODO: Höher stellen

// Axis Run
fbAxisLift.Enable := TRUE;
fbAxisLift.EnableCtrl := TRUE;
fbAxisLift.EnableNeg := TRUE;
fbAxisLift.EnablePos := TRUE;
fbAxisLift.Override := 100; //TODO: Höher stellen
fbAxisLift.TorqueLimit := 10; //TODO: Höher stellen

// Axis Run
fbAxisTelescope.Enable := TRUE;
fbAxisTelescope.EnableCtrl := TRUE;
fbAxisTelescope.EnableNeg := TRUE;
fbAxisTelescope.EnablePos := TRUE;
fbAxisTelescope.Override := 100; //TODO: Höher stellen
fbAxisTelescope.TorqueLimit := 10; //TODO: Höher stellen
END_METHOD

METHOD SetReferences : E_OperationResult
VAR_IN_OUT
	stIO				: ST_RackFeederIO;
END_VAR

VAR_INPUT
	Simulation			: BOOL;
END_VAR
bSimulation := Simulation;

fbAxisTraverse.SetReferences(stIO.ioAxisTraverse);
fbAxisTraverse.Name := 'Achse Traverse';
fbAxisTraverse.AxisType := E_AxisType.Virtual;
fbAxisTraverse.BMK := CONCAT3(THIS^.sName,' | ',fbAxisTraverse.Name);
{region "Default Parameter Traverse"}
fbAxisTraverse.DefaultParameter.stMovAbsPrm.fVelocity := 10;
fbAxisTraverse.DefaultParameter.stMovModPrm.fVelocity := 10;
fbAxisTraverse.DefaultParameter.stMovModPrm.eDirection := MC_Direction.MC_Shortest_Way;
fbAxisTraverse.DefaultParameter.stHomingPrm.fPosition := 0;
fbAxisTraverse.DefaultParameter.stHomingPrm.stOptions.SearchDirection := MC_Direction.MC_Positive_Direction;
fbAxisTraverse.DefaultParameter.stHomingPrm.stOptions.SearchVelocity := 10;
fbAxisTraverse.DefaultParameter.stHomingPrm.stOptions.SyncVelocity := 5;
fbAxisTraverse.DefaultParameter.stHomingPrm.stOptions.SyncDirection := MC_Direction.MC_Positive_Direction;
{endregion}

fbAxisLift.SetReferences(stIO.ioAxisLift);
fbAxisLift.Name := 'Achse Lift';
fbAxisLift.AxisType := E_AxisType.Virtual;
fbAxisLift.BMK := CONCAT3(THIS^.sName,' | ',fbAxisLift.Name);
{region "Default Parameter Lift"}
fbAxisLift.DefaultParameter.stMovAbsPrm.fVelocity := 10;
fbAxisLift.DefaultParameter.stMovModPrm.fVelocity := 10;
fbAxisLift.DefaultParameter.stMovModPrm.eDirection := MC_Direction.MC_Shortest_Way;
fbAxisLift.DefaultParameter.stHomingPrm.fPosition := 0;
fbAxisLift.DefaultParameter.stHomingPrm.stOptions.SearchDirection := MC_Direction.MC_Positive_Direction;
fbAxisLift.DefaultParameter.stHomingPrm.stOptions.SearchVelocity := 10;
fbAxisLift.DefaultParameter.stHomingPrm.stOptions.SyncVelocity := 5;
fbAxisLift.DefaultParameter.stHomingPrm.stOptions.SyncDirection := MC_Direction.MC_Positive_Direction;
{endregion}

fbAxisTelescope.SetReferences(stIO.ioAxisTelescope);
fbAxisTelescope.Name := 'Achse Telescope';
fbAxisTelescope.AxisType := E_AxisType.Virtual;
fbAxisTelescope.BMK := CONCAT3(THIS^.sName,' | ',fbAxisTelescope.Name);
{region "Default Parameter Telescope"}
fbAxisTelescope.DefaultParameter.stMovAbsPrm.fVelocity := 10;
fbAxisTelescope.DefaultParameter.stMovModPrm.fVelocity := 10;
fbAxisTelescope.DefaultParameter.stMovModPrm.eDirection := MC_Direction.MC_Shortest_Way;
fbAxisTelescope.DefaultParameter.stHomingPrm.fPosition := 0;
fbAxisTelescope.DefaultParameter.stHomingPrm.stOptions.SearchDirection := MC_Direction.MC_Positive_Direction;
fbAxisTelescope.DefaultParameter.stHomingPrm.stOptions.SearchVelocity := 10;
fbAxisTelescope.DefaultParameter.stHomingPrm.stOptions.SyncVelocity := 5;
fbAxisTelescope.DefaultParameter.stHomingPrm.stOptions.SyncDirection := MC_Direction.MC_Positive_Direction;
{endregion}

fbCarrierPresent.SetReferences(stIo.ioCarrierPresent);
END_METHOD

METHOD TeachStorageDock
VAR_IN_OUT
	Storage				: FB_Storage;
END_VAR
VAR_INPUT
	TeachPos				: BOOL;
END_VAR


VAR
	ni						: INT;
END_VAR
// Search if Reference is already in List
FOR ni := 0 TO nStorageDockCount DO

	IF NOT __ISVALIDREF(aTrolleyDocks[ni].refTrolley) THEN
		aStorageDocks[ni].refStorage REF= Storage;	
		EXIT;
	END_IF
	
	IF ADR(aStorageDocks[ni].refStorage) <> ADR(Storage) THEN
		CONTINUE;
	ELSE
		EXIT;
	END_IF

END_FOR


IF TeachPos THEN
// get Coordinate of Axis
	aStorageDocks[ni].posOrigin.fX := fbAxisTraverse.ActPos;
	aStorageDocks[ni].posOrigin.fY := fbAxisLift.ActPos;
	aStorageDocks[ni].posOrigin.fZ := fbAxisTelescope.ActPos;
	

	// set teched flag if Top an Buttom Value valid	
	aStorageDocks[ni].bTeached := TRUE;
END_IF
END_METHOD

METHOD TeachTrolleyDock
VAR_IN_OUT
	Trolley				: FB_Trolley;
END_VAR

VAR_INPUT
	TeachPosButtom			: BOOL;
	TeachPosTop				: BOOL;
END_VAR

VAR
	ni						: INT;
END_VAR
// Check Input
IF TeachPosButtom AND TeachPosTop THEN
	RETURN;
END_IF


// Search if Reference is already in List
FOR ni := 0 TO nTrolleyDockCount DO

	IF NOT __ISVALIDREF(aTrolleyDocks[ni].refTrolley) THEN
		aTrolleyDocks[ni].refTrolley REF= Trolley;	
		EXIT;
	END_IF
	
	IF ADR(aTrolleyDocks[ni].refTrolley) <> ADR(Trolley) THEN
		CONTINUE;
	ELSE
		EXIT;
	END_IF

END_FOR


// get Coordinate of Axis
IF TeachPosButtom THEN	
	aTrolleyDocks[ni].posButtom.fX := fbAxisTraverse.ActPos;
	aTrolleyDocks[ni].posButtom.fY := fbAxisLift.ActPos;
	aTrolleyDocks[ni].posButtom.fZ := fbAxisTelescope.ActPos;
	aTrolleyDocks[ni].bTeached := TRUE;
END_IF

IF TeachPosTop THEN
	aTrolleyDocks[ni].posTop.fX := fbAxisTraverse.ActPos;
	aTrolleyDocks[ni].posTop.fY := fbAxisLift.ActPos;
	aTrolleyDocks[ni].posTop.fZ := fbAxisTelescope.ActPos;
	aTrolleyDocks[ni].bTeached := TRUE;
END_IF


// set teched flag if Top an Buttom Value valid
END_METHOD

/// Visu component logic
{attribute 'object_name' := 'Visu'}
METHOD  Visu
CASE cmd.cmd OF
	E_RackFeederCmd.TeachTrolleyDock:
		;//TeachTrolleyDock(TRUE, TRUE, cmd.nId);
	
	E_RackFeederCmd.TeachStorageDock:
		;//TeachStorageDock(TRUE, TRUE);
	
		
END_CASE

IF cmd.cmd <> E_RackFeederCmd.noCmd THEN
	cmd.cmd := E_RackFeederCmd.noCmd; 
END_IF
END_METHOD

END_FUNCTION_BLOCK

// ---- Utilities/Component/FB_Component.TcPOU
/// Abstract base FB for components
{attribute 'reflection' := ''}
FUNCTION_BLOCK ABSTRACT FB_Component IMPLEMENTS ITF_Component

VAR
	/// path of this FB
	{attribute 'no_init' := ''}
	{attribute 'instance-path' := ''}
	sPath						: STRING;	
	/// Unique ID
	nId							: INT;		
	/// component type
	eTyp						: E_ComponentType;
	/// component name
	sName						: STRING;
	/// BMK name
	sBMK						: STRING;
	/// Area
	eMachineArea				: E_MachineArea;			
	
	/// component enable flag
	bEnable						: BOOL := FALSE;
	/// component state
	eState						: E_ComponentState;	
	
	/// Safety
	refEStop					: REFERENCE TO FB_EmergencyStop;
	aitfSafetyComp				: ARRAY[0..COMP.nMaxComponents] OF ITF_SafetyComp;
	bAccessPermit				: BOOL;


	/// Others
	itfEventLog					: ITF_EventLog;
	refSetting					: REFERENCE TO ST_MachineSetting;

	nChangeToggle				: INT;
END_VAR

///
/// 
/// HF/www.asma.at/02.2022
///

PROPERTY AccessPermit : BOOL
GET
AccessPermit := bAccessPermit;
END_GET
END_PROPERTY

/// RunSuper component logic
{attribute 'object_name' := 'Base'}
METHOD Base

VAR
	ni			: INT;
END_VAR
// DEFAULT STATE: set state to running
IF eState = E_ComponentState.ready THEN
	eState := E_ComponentState.running;
END_IF

//Eventlog
IF itfEventLog = 0 THEN
	WriteError(E_Event.eEvent_none, 'HMI Referenz nicht gesetzt!');
	eState := E_ComponentState.error;
	RETURN;
END_IF


Visu();

IF NOT Enable THEN
	RETURN;
END_IF

Run();
END_METHOD

PROPERTY BMK : STRING
GET
BMK := sBMK;
END_GET
SET
sBMK := BMK;
END_SET
END_PROPERTY

METHOD ChangeToggle : BOOL
VAR_INPUT
END_VAR
nChangeToggle := nChangeToggle + 1;
END_METHOD

PROPERTY EmergencyStop : REFERENCE TO FB_EmergencyStop
GET
IF __ISVALIDREF(refEStop) THEN
	EmergencyStop REF= refEStop;
END_IF
END_GET
SET
refEStop REF= EmergencyStop;
END_SET
END_PROPERTY

/// Get's or set's a value indicating whether this component is active or not.
PROPERTY Enable : BOOL
GET
Enable := bEnable;
END_GET
SET
bEnable := Enable;
END_SET
END_PROPERTY

METHOD FB_init : BOOL
VAR_INPUT
	bInitRetains : BOOL := TRUE; // if TRUE, the retain variables are initialized (warm start / cold start)
	bInCopyCode : BOOL := TRUE;  // if TRUE, the instance afterwards gets moved into the copy code (online change)
END_VAR
nId := nId + 1;
itfEventLog := GVL.fbEventLog;
refSetting REF= GVL.stSetting;
refEStop REF= GVL.fbEStop;
Init();
END_METHOD

/// Halt component logic
{attribute 'object_name' := 'Halt'}
METHOD Halt : E_OperationResult

VAR_INPUT
	StoppCategory					: INT;			// 0...ungesteuertes Stillsetzen     1...gesteuertes Stillsetzen     2...gesteuertes Stillsetzen ohne Trennung der Energiezufuhr							
END_VAR
bAccessPermit := TRUE;
END_METHOD

/// Unique component ID (cam be used as index: P_ComponentPool.aComponents[eID]...)
PROPERTY ID : INT
GET
ID := nId;
END_GET
SET
nId := Id;
END_SET
END_PROPERTY

/// Init component logic
{attribute 'object_name' := 'Init'}
METHOD Init : E_OperationResult
END_METHOD

PROPERTY MachineArea : E_MachineArea
GET
MachineArea := eMachineArea;
END_GET
SET
eMachineArea := MachineArea;
END_SET
END_PROPERTY

PROPERTY Name : STRING
GET
Name := sName;
END_GET
SET
sName := Name;
END_SET
END_PROPERTY

PROPERTY Path : String
GET
Path := sPath;
END_GET
END_PROPERTY

METHOD RegisterSafetyComp : BOOL
VAR_INPUT
	SafetyComp				: ITF_SafetyComp;
END_VAR
VAR
	ni						: INT;
END_VAR
FOR ni:= 0 TO COMP.nMaxComponents DO

	IF aitfSafetyComp[ni] = SafetyComp THEN
		RETURN;
	END_IF
	
	IF aitfSafetyComp[ni] <> 0 THEN
		CONTINUE;
	END_IF
	
	aitfSafetyComp[ni] := SafetyComp;
	aitfSafetyComp[ni].RegisterComponent(THIS^);
	RETURN;
	
END_FOR
END_METHOD

/// ResetSuper component logic
{attribute 'object_name' := 'Reset'}
METHOD Reset : E_OperationResult
// DEFAULT STATE: set state to ready
eState := E_ComponentState.ready;
END_METHOD

/// RestartSuper component logic
{attribute 'object_name' := 'Restart'}
METHOD Restart : E_OperationResult
VAR_INPUT
END_VAR
bAccessPermit := FALSE;
END_METHOD

/// RunSuper component logic
{attribute 'object_name' := 'Run'}
METHOD Abstract Run
END_METHOD

PROPERTY SafeEnvironment : BOOL
GET
VAR
	ni				: INT;
END_VAR
SafeEnvironment := TRUE;

FOR ni:= 0 TO COMP.nMaxComponents DO
	
	IF aitfSafetyComp[ni] <> 0 AND_THEN NOT aitfSafetyComp[ni].Safe THEN
		SafeEnvironment := FALSE;
	END_IF

END_FOR
END_GET
END_PROPERTY

/// Get's value representing the component state.
PROPERTY State : E_ComponentState
GET
State := eState;
END_GET
END_PROPERTY

/// Get's value representing the component state.
PROPERTY StateAsString : STRING
GET
CASE eState OF

	E_ComponentState.none :
		StateAsString := 'undefiniert';
	/// Component is resetting
	E_ComponentState.resetting:
		StateAsString := 'wird zurückgesetzt';
	/// Component is ready
	E_ComponentState.ready:
		StateAsString := 'ist bereit';
	/// Component is running
	E_ComponentState.running:
		StateAsString := 'wird ausgeführt';
	/// Component has error
	E_ComponentState.error:
		StateAsString := 'ist fehlerhaft';

END_CASE
END_GET
END_PROPERTY

PROPERTY Typ : E_ComponentType
GET
Typ := eTyp;
END_GET
END_PROPERTY

/// Visu component logic
{attribute 'object_name' := 'Visu'}
METHOD Abstract Visu
END_METHOD

METHOD VisuBase
VAR_IN_OUT
	stCompVisu					: ST_ComponentVisu;
END_VAR
// Visu
stCompVisu.bEnable := bEnable;
stCompVisu.bAccessPermit := AccessPermit;
stCompVisu.bError := eState = E_Componentstate.error;
stCompVisu.bRunning := eState = E_Componentstate.running;
stCompVisu.eState := eState;
stCompVisu.sName := sName;

IF stCompVisu.bReset THEN
	stCompVisu.bReset := FALSE;	
	Reset();
END_IF
END_METHOD

METHOD WriteError
VAR_INPUT
	Event			: E_Event;
	Description 	: T_MaxString;
END_VAR
WriteEvent(ePriority_fault, Event, Description, TRUE);
END_METHOD

METHOD WriteEvent
VAR_INPUT
	Priority		: E_Priority;
	Event			: E_Event;
	Description 	: T_MaxString;
	Signalize		: BOOL;
END_VAR
VAR
	tmpItem: ST_Event;
END_VAR
// chk
IF itfEventLog = 0 THEN
	RETURN;
END_IF

tmpItem.eComponent := eTyp;
tmpItem.eEventID := Event;
tmpItem.eMachineArea := eMachineArea;
tmpItem.sPosition := sBMK;
tmpItem.ePriority := Priority;
tmpItem.nComponentID := nId;
tmpItem.sDescription := Description;
tmpItem.bSignalize := Signalize;
tmpItem.refComponent REF= THIS^;

itfEventLog.SetEvent(tmpItem);
END_METHOD

METHOD WriteInfo
VAR_INPUT
	Event			: E_Event;
	Description 	: T_MaxString;
END_VAR
WriteEvent(ePriority_info, Event, Description, FALSE);
END_METHOD

METHOD WriteWarning
VAR_INPUT
	Event			: E_Event;
	Description 	: T_MaxString;
	Signal			: BOOL;
END_VAR
VAR
	tmpItem			: ST_Event;
END_VAR
WriteEvent(ePriority_warning, Event, Description, Signal);
END_METHOD

END_FUNCTION_BLOCK

// ---- Template/Station/ST001.TcPOU
FUNCTION_BLOCK ST001 EXTENDS TcoCore.TcoObject
VAR	
	{attribute addProperty Name "<#MANUAL#>"}
	_serviceModeTask : TcoCore.TcoTask(THIS^);
    {attribute addProperty Name "<#GROUND#>"}	
	_groundSequenceTask  : TcoCore.TcoTask(THIS^);
	{attribute addProperty Name "<#AUTOMAT#>"}	
	_automatSequenceTask  : TcoCore.TcoTask(THIS^);
	
	{attribute clr [Container(Layout.Stack)]}
	_components : ST001_ComponentsHandler(THIS^);
	
	{attribute clr [RenderIgnore()]}
	_mqttMirrorComponents : ST001_ComponentsHandler(THIS^);
	
	{attribute clr [Container(Layout.Stack)]}
	_groundPositionSequence : ST001_GroundSequence(THIS^, eRestoreMode.None);
	_automatPositionSequence : ST001_AutomatSequence(THIS^, eRestoreMode.None);
	
	_settings 	: ST001_ProcessDataManager(THIS^);
	_repository : ST001_ProcessDataManager(THIS^);
END_VAR

_components();
_settings();
_repository();
_groundPositionSequence(inoComponents := _components);
_automatPositionSequence(inoComponents := _components);


IF(_groundSequenceTask.Execute()) THEN
	_serviceModeTask.Abort();
	_groundPositionSequence.Run();
	_groundSequenceTask.DoneWhen(_groundPositionSequence.CurrentStep.ID = _groundPositionSequence.MaxStepID - 1);	
END_IF

_automatSequenceTask.Enabled := _groundSequenceTask.Done;

IF(_automatSequenceTask.Execute()) THEN	
	_automatPositionSequence.Run();
END_IF

IF(_serviceModeTask.Execute()) THEN
	_automatSequenceTask.Restore();	
	_groundSequenceTask.Restore();
	_groundPositionSequence.Restore();
	_components.Service();
END_IF

PROPERTY Repository : REFERENCE TO ST001_ProcessDataManager
GET
Repository REF= _repository;
END_GET
END_PROPERTY

PROPERTY Settings : REFERENCE TO ST001_ProcessDataManager
GET
Settings REF= _settings;
END_GET
END_PROPERTY

END_FUNCTION_BLOCK

// ---- Template/Station/ST001_ComponentsHandler.TcPOU
FUNCTION_BLOCK ST001_ComponentsHandler EXTENDS TcoCore.TcoObject
VAR
	ToMirror:STRING;
	{attribute addProperty Name "<#PART PRESENCE SENSOR#>"}
	_partPresent : TcoElements.TcoDi(THIS^);
	{attribute addProperty Name "<#START BUTTON#>"}
    _startButton : TcoElements.TcoDi(THIS^);
	{attribute addProperty Name "<#PRESS PISTON#>"}
    _press : TcoPneumatics.TcoCylinder(THIS^);
	{attribute addProperty Name "<#ALARM OUTPUT#>"}
	_alarmOutput : TcoElements.TcoDo(THIS^);
	{attribute addProperty Name "<#DRIVE#>"}
	_drive : TcoDrivesBeckhoff.TcoDriveSimple(THIS^);
END_VAR

_partPresent(inoSignal := IO.EC001.A1.IO._1);
_startButton(inoSignal := IO.EC001.A1.IO._2);
_press(inoAtHomePos:= IO.EC001.A1.IO._3, inoAtWorkPos:= IO.EC001.A1.IO._4, inoToHomePos:= IO.EC001.A10.IO._1, inoToWorkPos:=IO.EC001.A10.IO._2);

PROPERTY PartPresent : REFERENCE TO TcoElements.TcoDi
GET
PartPresent REF= _partPresent;
END_GET
END_PROPERTY

PROPERTY Press : REFERENCE TO TcoPneumatics.TcoCylinder
GET
Press REF= _press;
END_GET
END_PROPERTY

METHOD Service
THIS^._partPresent.Service();
THIS^._startButton.Service();
THIS^._press.Service();
THIS^._alarmOutput.Service();
END_METHOD

END_FUNCTION_BLOCK

// ---- Template/Station/ST001_GroundSequence.TcPOU
FUNCTION_BLOCK ST001_GroundSequence EXTENDS TcoCore.TcoSequencer
VAR_IN_OUT
	inoComponents : ST001_ComponentsHandler;
END_VAR

(*~
	<docu>
		<summary>
			Main method of the sequener. Custom code needs to be placed here. The sequencer is executed by call of InstanceName.Run() method.
			This method is abstract, and it must be overridden in derived block.
		</summary>
	</docu>
~*)
METHOD PROTECTED  Main : BOOL
IF(NOT __ISVALIDREF(inoComponents)) THEN
	Messenger.Programming('Invalid reference to inoComponents');
	RETURN;
END_IF


IF(Step(inStepID  			:= 100,
	    inEnabled 			:= TRUE,
	    inStepDescription 	:= '<#PRESS IN BASE POSITION#>')) 
THEN
//---------------------------------------
	IF(inoComponents.Press.MoveToHome().Done) THEN
		THIS^.CompleteStep();		
	END_IF;
//---------------------------------------
END_IF;

IF(Step(inStepID  			:= 200,
	    inEnabled 			:= TRUE,
	    inStepDescription 	:= '<#CHECK PART REMOVAL FROM THE FIXTURE#>')) 
THEN
//---------------------------------------
	IF(inoComponents.PartPresent.IsFalse) THEN
		THIS^.CompleteStep();
	ELSE
		Messenger.Notify('<#Remove part from the fixture please#>');	
	END_IF;
//---------------------------------------
END_IF;

IF(Step(inStepID  			:= MaxStepID - 1,
	    inEnabled 			:= TRUE,
	    inStepDescription 	:= '<#GROUND POSITION COMPLETED#>')) 
THEN
//---------------------------------------
	Messenger.Notify('<#Ground position completed; you can start automat sequence.#>');	
//---------------------------------------
END_IF;
END_METHOD

METHOD PROTECTED OnStateChange
VAR_INPUT
	PreviousState	: INT;
	NewState 		: INT;
END_VAR
IF(NOT __ISVALIDREF(inoComponents)) THEN
	RETURN;
END_IF

inoComponents.Press.Restore();
END_METHOD

END_FUNCTION_BLOCK

// ---- Template/Component_Carousell/Tasks/TcoTurnTableTask.TcPOU
FUNCTION_BLOCK TcoTurnTableTask EXTENDS TcoCore.TcoTask
VAR_INPUT
	inSafetyCondition:BOOL;
END_VAR
VAR_IN_OUT

	inoInPosition : BOOL;
	inoInPrecisePosition : BOOL;
	inoEnableTurn : BOOL;
	inoStartTurn : BOOL;
	inoConfig : TcoCarouselConfig;
	inoStatus : TcoCarouselStatus;
END_VAR

VAR
 	{attribute 'hide'} 
	_progress : INT := 0;
    {attribute 'hide'} 
	_infoTimer :  TON;
    {attribute 'hide'} 
	_errorTimer :  TON;
    {attribute 'hide'} 
	_varInfo : __SYSTEM.VAR_INFO;
    {attribute 'hide'} 
	_sb : TcoCore.StringBuilder;
	
	_notInPositionMessage : TcoCore.TcoMessenger(THIS^);	
END_VAR

IF (THIS^.Execute()) THEN


	IF _progress = 0 THEN
		IF NOT __ISVALIDREF(inoInPosition) THEN
			_varInfo :=__VARINFO(inoInPosition);
			Messenger.Programming(_sb.Clear().Append('<#Invalid reference: #>').Append(_varInfo.Symbol).ToString()).Pin();
		ELSIF NOT __ISVALIDREF(inoInPrecisePosition) THEN                                              
			_varInfo :=__VARINFO(inoInPrecisePosition);                                                
			Messenger.Programming(_sb.Clear().Append('<#Invalid reference: #>').Append(_varInfo.Symbol).ToString()).Pin();
		ELSIF NOT __ISVALIDREF(inoEnableTurn) THEN                                              
			_varInfo :=__VARINFO(inoEnableTurn);                                                
			Messenger.Programming(_sb.Clear().Append('<#Invalid reference: #>').Append(_varInfo.Symbol).ToString()).Pin();
		ELSIF NOT __ISVALIDREF(inoStartTurn) THEN                                              
			_varInfo :=__VARINFO(inoStartTurn);                                                
			Messenger.Programming(_sb.Clear().Append('<#Invalid reference: #>').Append(_varInfo.Symbol).ToString()).Pin();
		ELSIF NOT __ISVALIDREF(inoConfig) THEN                                                  
			_varInfo :=__VARINFO(inoConfig);                                                    
			Messenger.Programming(_sb.Clear().Append('<#Invalid reference: #>').Append(_varInfo.Symbol).ToString()).Pin();
		ELSIF NOT __ISVALIDREF(inoStatus) THEN                                                  
			_varInfo :=__VARINFO(inoStatus);                                                    
			Messenger.Programming(_sb.Clear().Append('<#Invalid reference: #>').Append(_varInfo.Symbol).ToString()).Pin();
	
		ELSE
			_progress := _progress + 1;
		END_IF

	END_IF
	IF _progress=1 THEN	
		_notInPositionMessage.OnCondition(NOT inoInPosition).Error('<#Rotatiting started , but table is not in default position! Acknowledge this alarm if you still want to turn! #>').Pin();
		_progress:=10;
	
	END_IF;
	

	
	IF _progress=10 THEN	
		Messenger.Info('<#Calulate next expected Id position#>');
		IF inoStatus.CurrentPosition <> 0 THEN
			inoStatus.ExpectedNextPosition := GetIdentifierAtPosition( inoConfig.NumberOfPositions,inoStatus.Positions);	
		END_IF;
		
		Messenger.OnCondition(inoStatus.CurrentPosition=0  AND inoInPosition).Error('<#Incorrectly coded current position. Check configuration of code bits! #>').Pin();
		
		IF	inoStatus.CurrentPosition <> 0 AND inoInPosition THEN
			_progress := 20;
		ELSIF NOT 	_notInPositionMessage.Pinned THEN
			_progress:=20;
			_notInPositionMessage.UnPin();
	
		END_IF;		
	END_IF;
	
	IF _progress=20 THEN	
		inoEnableTurn:=TRUE; 
		inoStartTurn:=TRUE;	
		Messenger.Info('<#Table turning. Trying to leave sensor#>');
		
		IF NOT inoInPosition THEN
			inoEnableTurn:=FALSE;	
			_progress :=  _progress+10;				
		END_IF
	END_IF;
	
	
	IF _progress=30 THEN	
		Messenger.Info('<#Table turning. Trying to reach sensor table in positon.#>');
		inoStartTurn:=TRUE;	
		IF inoInPosition THEN
			inoEnableTurn:=FALSE; 
			inoStartTurn:=FALSE;	
			_progress :=  _progress+10;				
		END_IF
	END_IF;
	
	IF _progress=40 THEN	
		Messenger.OnCondition(inoStatus.CurrentPosition > 0 AND_THEN inoStatus.ExpectedNextPosition  <>  GetIdentifierAtPosition(1,inoStatus.Positions)).
			Error(_sb.Clear().Append('<#Table after turn does not have expected coding. Expected id at position #1 is#> ').Append( UINT_TO_STRING(inoStatus.ExpectedNextPosition)).ToString()).Pin();
	
		IF(inoStatus.CurrentPosition > 0 AND inoStatus.ExpectedNextPosition = GetIdentifierAtPosition(1,inoStatus.Positions)) THEN
			
			THIS^.DoneWhen(TRUE);	
	
		END_IF;	
	END_IF;
	
	
	CallTimers(TRUE);
	THIS^.ThrowWhen(_errorTimer.Q);	
	
END_IF


IF NOT inSafetyCondition THEN
	inoEnableTurn:=FALSE; 
	inoStartTurn:=FALSE;	
	Messenger.Error('<#Safety conditions to turn the table are not met.#>').Pin();
END_IF

METHOD CallTimers
VAR_INPUT
	inValue : BOOL;
END_VAR
IF  __ISVALIDREF(inoConfig) THEN  
_infoTimer(IN := inValue, PT := THIS^.inoConfig.InfoTime);
_errorTimer(IN := inValue, PT := THIS^.inoConfig.ErrorTime);
END_IF;
END_METHOD

{attribute 'hide'}
METHOD PUBLIC FB_init : BOOL
VAR_INPUT
	bInitRetains : BOOL; // if TRUE, the retain variables are initialized (warm start / cold start)
	bInCopyCode : BOOL;  // if TRUE, the instance afterwards gets moved into the copy code (online change)
	ParentObject : ITcoObject;
END_VAR
END_METHOD

METHOD  GetIdentifierAtPosition : UINT
VAR_INPUT
	inPosition : UINT;
	inPositions : ARRAY[0..20] OF UINT;
END_VAR
IF(inPosition < 1 OR inPosition >  SIZEOF (inPositions)) THEN
	Messenger.Programming(Concat('<#Required position must be in range 1 - 20 but was:#>', UINT_TO_STRING(inPosition)));
	RETURN;
END_IF

GetIdentifierAtPosition := inPositions[inPosition - 1];
END_METHOD

(*~
	<docu>
		<summary>
			Executes when task is aborted.
		</summary>			
	</docu>	
~*)
METHOD PROTECTED OnAbort
IF  __ISVALIDREF(inoStatus) THEN   THIS^.inoStatus.ActionDescription := '<#Turning table was aborted, while not yet completed!#>';END_IF;
END_METHOD

(*~
	<docu>
		<summary>
			Executes when task reaches the ```Done``` state .
		</summary>			
	</docu>	
~*)
METHOD PROTECTED OnDone
IF  __ISVALIDREF(inoStatus) THEN  THIS^.inoStatus.ActionDescription := '<#Truning table  was completed successfully.#>';END_IF;
END_METHOD

METHOD PROTECTED OnError
IF  __ISVALIDREF(inoStatus) THEN   THIS^.inoStatus.ActionDescription := '<#Turning table finished with an error.#>'; END_IF;
END_METHOD

METHOD PROTECTED OnStart
IF  __ISVALIDREF(inoStatus) THEN  THIS^.inoStatus.ActionDescription := '<#Turning table started.#>'; END_IF;
END_METHOD

(*~
	<docu>
		<summary>
			Restores this instance to the Ready state. Can be called explicitly or from within one of the restore mechanisms.
			<para>
				See also <see cref="PlcDocu.TcoCore.TcoTask.AutoRestorable()"/>
			</para>
		</summary>			
	</docu>	
~*)
METHOD Restore : ITcoRestorable
SUPER^.Restore();
_progress := 0;
CallTimers(FALSE);
Messenger.UnPin();
_notInPositionMessage.UnPin();
END_METHOD

END_FUNCTION_BLOCK

// ---- Utilities/EventLog/FB_EventLog.TcPOU
/// HMI access provider (host for sub hmi provider)
FUNCTION_BLOCK  FB_EventLog IMPLEMENTS ITF_EventLog

VAR		
	stVisu						: ST_EventVisu;
	
	aRaisedEvents				: ARRAY[0..nMaxEvents] OF ST_Event;
	aQuitEvents					: ARRAY[0..nMaxEvents] OF ST_Event;

	
	eLogLevel					: E_LogLevel;	
	bMute						: BOOL;

	nErrorCount					: INT;
	nWarningCount				: INT;
	nInfoCount					: INT;
	
END_VAR

///
/// Event Log
/// Hannes Fuger /www.asma.at/01.2016
///

PROPERTY ErrorCount : INT
GET
ErrorCount := nErrorCount;
END_GET
END_PROPERTY

/// System error level
PROPERTY ErrorLevel : E_Priority
GET // INTERNAL
VAR
	ni			: INT;
END_VAR
FOR ni:= 0 TO nMaxEvents DO
	
	IF aRaisedEvents[ni].ePriority = E_Priority.ePriority_none OR ErrorLevel = E_Priority.ePriority_faultEmergency THEN
		RETURN;
	END_IF

	ErrorLevel := MAX(ErrorLevel, aRaisedEvents[ni].ePriority);
	
END_FOR
END_GET
END_PROPERTY

PROPERTY InfoCount : INT
GET
InfoCount := nInfoCount;
END_GET
END_PROPERTY

PROPERTY LogLevel : E_LogLevel
GET
LogLevel := eLogLevel;
END_GET
SET
eLogLevel := LogLevel;
END_SET
END_PROPERTY

PROPERTY Mute : BOOL
GET
Mute := bMute;
END_GET
SET
bMute := Mute;
END_SET
END_PROPERTY

/// sets the corresponding notification item flag raised
{attribute 'object_name' := 'Quitt'}
METHOD Quitt
VAR_INPUT
	Index			: INT;
END_VAR
VAR
	ni				: INT;
	cmpEvent		: ST_Event;
END_VAR
CASE aRaisedEvents[Index].ePriority OF
	
	E_Priority.ePriority_fault, E_Priority.ePriority_faultEmergency, E_Priority.ePriority_faultFastStop:
		nErrorCount := nErrorCount - 1;
	
	E_Priority.ePriority_info:
		nInfoCount := nInfoCount - 1;
	
	E_Priority.ePriority_warning:
		nWarningCount := nWarningCount - 1;

END_CASE

// Reset Component
IF __ISVALIDREF(aRaisedEvents[Index].refComponent) THEN
	aRaisedEvents[Index].refComponent.Reset();
END_IF

// Copy Event from Raised to Quit Table
MEMMOVE(ADR(aQuitEvents[1]), ADR(aQuitEvents[0]), TO_UDINT(nMaxEvents-1)*SIZEOF(aQuitEvents[1]));
aQuitEvents[0] := aRaisedEvents[Index];
aQuitEvents[0].dtQuitTime := Statics.dtNow;	


// Delete Event from Raised Table
MEMMOVE(ADR(aRaisedEvents[Index]), ADR(aRaisedEvents[Index+1]), TO_UDINT(nMaxEvents-Index)*SIZEOF(aRaisedEvents[Index]));
END_METHOD

/// sets the corresponding notification item flag raised
{attribute 'object_name' := 'QuittAll'}
METHOD QuittAll
VAR_INPUT
	eMachineArea	: E_MachineArea;
END_VAR
VAR
	ni				: INT;
END_VAR
FOR ni := 0 TO nMaxEvents DO	
	
	IF aRaisedEvents[0].ePriority = E_Priority.ePriority_none THEN
		RETURN;
	END_IF
	
	IF aRaisedEvents[0].eMachineArea = eMachineArea OR eMachineArea = E_MachineArea.none THEN
		Quitt(0);
	END_IF
	
END_FOR
END_METHOD

/// sets the corresponding notification item flag raised
{attribute 'object_name' := 'QuittEvent'}
METHOD QuittEvent
VAR_INPUT
	stEvent			: ST_Event;
END_VAR
VAR
	ni				: INT;
	cmpEvent		: ST_Event;
END_VAR
cmpEvent := stEvent;

FOR ni := 0 TO nMaxEvents DO	
			
	IF MEMCMP(ADR(cmpEvent), ADR(aRaisedEvents[ni]), SIZEOF(St_EventBase)) = 0 THEN
		
		// Copy Event from Raised to Quit Table
		MEMMOVE(ADR(aQuitEvents[1]), ADR(aQuitEvents[0]), TO_UDINT(nMaxEvents-1)*SIZEOF(ST_Event));
		aQuitEvents[0] := aRaisedEvents[ni];
		aQuitEvents[0].dtQuitTime := Statics.dtNow;	

		// Delete Event from Raised Table
		MEMMOVE(ADR(aRaisedEvents[ni]), ADR(aRaisedEvents[ni+1]), TO_UDINT(nMaxEvents-ni)*SIZEOF(ST_Event));
	
	END_IF
	
END_FOR
END_METHOD

/// resets all notification flags and reset-needed state 
{attribute '' := ''}
{attribute 'object_name' := 'Reset'}
METHOD Reset
VAR
	ResetEvent	: st_Event;
	ii: INT;
END_VAR
// reset all items in default notification array
MEMSET(ADR(aRaisedEvents), 0, SIZEOF(aRaisedEvents));
MEMSET(ADR(aQuitEvents), 0, SIZEOF(aQuitEvents));

nErrorCount		:= 0;
nWarningCount	:= 0;
nInfoCount		:= 0;

eLogLevel			:= eLogLevelInformation;
END_METHOD

METHOD Run
VAR	/// private variabe
	ii			: INT;	
END_VAR
Visu();
END_METHOD

/// sets the corresponding notification item flag raised
{attribute 'object_name' := 'SetEvent'}
METHOD SetEvent 
VAR_INPUT
	/// item to set
	stEvent			: ST_Event;
END_VAR

VAR
	ni				: INT;
	cmpEvent		: ST_EventBase;
	presentEvent	: ST_EventBase;
END_VAR
IF TO_INT(stEvent.ePriority) < TO_INT(eLogLevel) THEN
	RETURN;
END_IF

IF stEvent.eEventID = E_Event.eEvent_none THEN

	IF 	stEvent.ePriority = E_Priority.ePriority_fault OR stEvent.ePriority = E_Priority.ePriority_faultEmergency OR stEvent.ePriority = E_Priority.ePriority_faultFastStop THEN
		stEvent.eEventID := E_Event.eEvent_generalError;
	ELSIF 	stEvent.ePriority = E_Priority.ePriority_warning THEN
		stEvent.eEventID := E_Event.eEvent_generalWarning;
	ELSIF 	stEvent.ePriority = E_Priority.ePriority_info THEN
		stEvent.eEventID := E_Event.eEvent_generalInfo;
	END_IF 
	
END_IF

cmpEvent := stEvent;

// look for Same Event
FOR ni:=0 TO nMaxEvents DO
	
	// Event not in List
	IF aRaisedEvents[ni].ePriority = E_Priority.ePriority_none THEN
		EXIT;
	END_IF
	
	presentEvent := aRaisedEvents[ni];
	
	// Same Event in List
	IF 	presentEvent.eComponent = 	cmpEvent.eComponent AND_THEN
		presentEvent.ePriority = 	cmpEvent.ePriority AND_THEN 
		presentEvent.nComponentID = cmpEvent.nComponentID AND_THEN
		//ADR(presentEvent.refComponent) = ADR(cmpEvent.refComponent) AND_THEN 
		presentEvent.sDescription = cmpEvent.sDescription AND_THEN
		presentEvent.eEventID =     cmpEvent.eEventID AND_THEN
		presentEvent.bSignalize =   cmpEvent.bSignalize AND_THEN
		presentEvent.sPosition =    cmpEvent.sPosition AND_THEN
		presentEvent.eMachineArea = cmpEvent.eMachineArea THEN
		
			// insert new Event on First Place
			MEMMOVE(ADR(aRaisedEvents[1]), ADR(aRaisedEvents[0]), TO_UDINT(ni)*SIZEOF(stEvent));
			aRaisedEvents[0] := stEvent;
			aRaisedEvents[0].dtRaiseTime := Statics.dtNow;
			RETURN;
			
	END_IF

	
END_FOR


// insert new Event on First Place
MEMMOVE(ADR(aRaisedEvents[1]), ADR(aRaisedEvents[0]), TO_UDINT(nMaxEvents-1)*SIZEOF(stEvent));
aRaisedEvents[0] := stEvent;
aRaisedEvents[0].dtRaiseTime := Statics.dtNow;

CASE aRaisedEvents[0].ePriority OF
	
	E_Priority.ePriority_fault, E_Priority.ePriority_faultEmergency, E_Priority.ePriority_faultFastStop:
		nErrorCount := nErrorCount + 1;
	
	E_Priority.ePriority_info:
		nInfoCount := nInfoCount + 1;
	
	E_Priority.ePriority_warning:
		nWarningCount := nWarningCount + 1;

END_CASE
END_METHOD

METHOD UcControl : BOOL
VAR_IN_OUT
	stVisu			: Uc_EventLogControl;
END_VAR
stVisu.nErrorCount		:= nErrorCount;
stVisu.nWarningCount	:= nWarningCount;
stVisu.nInfoCount		:= nInfoCount;

stVisu.nErrorColor 		:= colEventError;
stVisu.nWarningColor 	:= colEventWarning;	
stVisu.nInfoColor 		:= colEventInfo;	

IF stVisu.bQuittAll THEN
	stVisu.bQuittAll := FALSE;
	QuittAll(E_MachineArea.none);
END_IF
END_METHOD

METHOD UcTable : BOOL
VAR_IN_OUT
	stVisu				: Uc_EventLogTable;
	stControl			: Uc_EventLogControl;
END_VAR

VAR
	ni					: INT;
	nj					: INT;
END_VAR

VAR_INST
	aOldRaisedEvents	: ARRAY[0..nMaxEvents] OF ST_Event;
	RESULT				: ARRAY[0..nMaxEvents] OF ST_EventOutput;		
END_VAR
IF stVisu.bQuitt THEN
	stVisu.bQuitt := FALSE;
	Quitt(stVisu.nIdx);
END_IF


IF MEMCMP(ADR(aRaisedEvents), ADR(aOldRaisedEvents), SIZEOF(aRaisedEvents)) = 0 AND NOT stControl.bFilterChanged THEN
	RETURN;
END_IF

stControl.bFilterChanged := FALSE;

MEMCPY(ADR(aOldRaisedEvents), ADR(aRaisedEvents), SIZEOF(aRaisedEvents));
MEMSET(ADR(stVisu.astEvents), 0, SIZEOF(stVisu.astEvents));

FOR nj:=0 TO nMaxEvents DO
	stVisu.astEvents[nj].nIdx := -1;	
END_FOR

nj:=0;

FOR ni:=0 TO nMaxEvents DO

		// FILTER
		IF aRaisedEvents[ni].ePriority = ePriority_none THEN
			CONTINUE;
		END_IF
	
		IF NOT stControl.bErrorFilter AND aRaisedEvents[ni].ePriority = E_Priority.ePriority_fault THEN
			CONTINUE;
		END_IF
		
		IF NOT stControl.bErrorFilter AND aRaisedEvents[ni].ePriority = E_Priority.ePriority_faultEmergency THEN
			CONTINUE;
		END_IF
		
		IF NOT stControl.bErrorFilter AND aRaisedEvents[ni].ePriority = E_Priority.ePriority_faultFastStop THEN
			CONTINUE;
		END_IF
		
		IF NOT stControl.bWarningFilter AND aRaisedEvents[ni].ePriority = E_Priority.ePriority_warning THEN
			CONTINUE;
		END_IF
		
		IF NOT stControl.bInfoFilter AND aRaisedEvents[ni].ePriority = E_Priority.ePriority_info THEN
			CONTINUE;
		END_IF
		
		IF stControl.eAreaFilter <> E_MachineArea.None AND aRaisedEvents[ni].eMachineArea <> stControl.eAreaFilter THEN
			CONTINUE;
		END_IF
		
		
		// add notification to result
		stVisu.astEvents[nj].sDescription := aRaisedEvents[ni].sDescription;
		stVisu.astEvents[nj].sPosition := aRaisedEvents[ni].sPosition;
		stVisu.astEvents[nj].sRaiseInfo := CONCAT3(TO_STRING(aRaisedEvents[ni].eEventID),' | ',  F_DT_TO_STRING(aRaisedEvents[ni].dtRaiseTime));	
		stVisu.astEvents[nj].nIdx := ni;
		
		CASE  aRaisedEvents[ni].ePriority OF
			
			ePriority_none :
				stVisu.astEvents[nj].nPriorityColor := colEventNone;
				stVisu.astEvents[nj].sPriority := "";				
			ePriority_info :
				stVisu.astEvents[nj].nPriorityColor := colEventInfo;
				stVisu.astEvents[nj].sPriority := "ℹ";
			ePriority_warning :
				stVisu.astEvents[nj].nPriorityColor := colEventWarning;
				stVisu.astEvents[nj].sPriority := "⚠";
			ePriority_fault :
				stVisu.astEvents[nj].nPriorityColor := colEventError;
				stVisu.astEvents[nj].sPriority := "❎";
			ePriority_faultFastStop :
				stVisu.astEvents[nj].nPriorityColor := colEventError;
				stVisu.astEvents[nj].sPriority := "❎";
			ePriority_faultEmergency :
				stVisu.astEvents[nj].nPriorityColor := colEventError;
				stVisu.astEvents[nj].sPriority := "❌";
			
		END_CASE
		
		nj := nj + 1;	
		
END_FOR
END_METHOD

METHOD Visu
VAR_INPUT
END_VAR
UcControl(stVisu.ucControl);
UcTable(stVisu.ucTable, stVisu.ucControl);
END_METHOD

PROPERTY WarningCount : INT
GET
WarningCount := nWarningCount;
END_GET
END_PROPERTY

END_FUNCTION_BLOCK

// ---- Utilities/Helpers/F_DT_TO_STRING.TcPOU
FUNCTION F_DT_TO_STRING : STRING
VAR_INPUT
	dtTime			: DT;
END_VAR
VAR
	timeStruct		: TIMESTRUCT;
END_VAR

F_DT_TO_STRING := SYSTEMTIME_TO_STRING(DT_TO_SYSTEMTIME(dtTime));

//F_DT_TO_STRING := CONCAT6(F_TO_STRING(timeStruct.wDay), '.', F_TO_STRING(timeStruct.wMonth), '.', F_TO_STRING(timeStruct.wYear), ' - ');
//F_DT_TO_STRING := CONCAT6(F_DT_TO_STRING, F_TO_STRING(timeStruct.wHour), ':', F_TO_STRING(timeStruct.wMinute), ':', F_TO_STRING(timeStruct.wSecond));

END_FUNCTION

// ---- Utilities/Helpers/Color/F_DWORD2RGB.TcPOU
FUNCTION F_DWORD2RGB : ST_Color
VAR_INPUT
	Color					: DWORD;
END_VAR

VAR
	tmpArray				: ARRAY[0..3] OF BYTE;
END_VAR

MEMCPY(ADR(tmpArray), ADR(Color), SIZEOF(DWORD));

F_DWORD2RGB.nTransparency := tmpArray[3];
F_DWORD2RGB.nRed := tmpArray[2];
F_DWORD2RGB.nGreen := tmpArray[1];
F_DWORD2RGB.nBlue := tmpArray[0];

END_FUNCTION

// ---- Utilities/Helpers/Color/F_RGB2CMYK.TcPOU
FUNCTION F_RGB2CMYK : ST_ColorCMYK
VAR_INPUT
	Color					: ST_Color;
END_VAR

VAR
	stColor					: ST_COLOR;
	tmpArray				: ARRAY[0..3] OF BYTE;
	
	Rc						: REAL;
	Gc						: REAL;
	Bc						: REAL;

	K						: REAL;
	
END_VAR

stColor := Color;

Rc := stColor.nRed / 255;
Gc := stColor.nGreen / 255;
Bc := stColor.nBlue / 255;

IF (Rc + Gc + Bc) = 0 THEN
	F_RGB2CMYK.nCyan := 0;
	F_RGB2CMYK.nMagenta := 0;
	F_RGB2CMYK.nYellow := 0;
	F_RGB2CMYK.nKey := 100;	
	RETURN;
END_IF

K := TO_BYTE(1 - MAX(Rc, MAX(Gc, Bc)));

F_RGB2CMYK.nCyan := TO_BYTE((1-Rc-K)/(1-K));
F_RGB2CMYK.nMagenta := TO_BYTE((1-Gc-K)/(1-K));
F_RGB2CMYK.nYellow := TO_BYTE((1-Bc-K)/(1-K));
F_RGB2CMYK.nKey := TO_BYTE(K);

END_FUNCTION

// ---- Utilities/Helpers/Color/F_TextColor.TcPOU
FUNCTION F_TextColor : DWORD
VAR_INPUT
	Color					: DWORD;
END_VAR

VAR
	stColor					: ST_COLOR;
	stWhite					: ST_COLOR;		
	stBlack					: ST_COLOR;			
	
	lblColorDifference		: INT;
	lblBrightnessDifference : UINT;
	
	
tmpArray				: ARRAY[0..3] OF BYTE;
	
	Rc						: INT;
	Gc						: INT;
	Bc						: INT;

	K						: INT;
	
END_VAR

stColor := F_DWORD2RGB(Color);
stWhite := F_DWORD2RGB(colWhite);
stBlack := F_DWORD2RGB(colBlack);

lblBrightnessDifference := (299*stColor.nRed + 587*stColor.nGreen + 114*stColor.nBlue)/1000 - (299*stWhite.nRed + 587*stWhite.nGreen + 114*stWhite.nBlue)/1000;
lblColorDifference := -((stColor.nRed - stWhite.nRed) + (stColor.nGreen - stWhite.nGreen + (stColor.nBlue - stWhite.nBlue)));

IF lblBrightnessDifference > 125 AND lblColorDifference > 500 THEN
	F_TextColor := colWhite;	
ELSE
	F_TextColor := colBlack;
END_IF

END_FUNCTION

// ---- Utilities/Helpers/Concat/Concat2.TcPOU
FUNCTION Concat2 : T_MaxString
VAR_INPUT
	sExpression1: T_maxString;
	sExpression2: T_maxString;
END_VAR

Concat2 := CONCAT(sExpression1, sExpression2);

END_FUNCTION

// ---- Utilities/Helpers/Concat/Concat7.TcPOU
FUNCTION Concat7 : T_MaxString
VAR_INPUT
	sExpression1: T_maxString;
	sExpression2: T_maxString;
	sExpression3: T_maxString;
	sExpression4: T_maxString;
	sExpression5: T_maxString;
	sExpression6: T_maxString;
	sExpression7: T_maxString;
END_VAR

Concat7 := CONCAT(sExpression1, sExpression2);
Concat7 := CONCAT(Concat7, sExpression3);
Concat7 := CONCAT(Concat7, sExpression4);
Concat7 := CONCAT(Concat7, sExpression5);
Concat7 := CONCAT(Concat7, sExpression6);
Concat7 := CONCAT(Concat7, sExpression7);

END_FUNCTION

// ---- Utilities/Helpers/F_BYTE_TO_REAL.TcPOU
FUNCTION F_BYTE_TO_REAL : REAL
VAR_INPUT
    BY1 : BYTE;
    BY2 : BYTE;
    BY3 : BYTE;
    BY4 : BYTE;
END_VAR
VAR
   OutVAR : DWORD; 
   OutVarREAL : REAL;
END_VAR

OutVar := BY1;
OutVar := SHL(OutVar, 8) OR BY2;
OutVar := SHL(OutVar, 8) OR BY3;
OutVar := SHL(OutVar, 8) OR BY4;

MEMCPY(ADR(OutVarREAL), ADR(OutVar), SIZEOF(REAL));
F_BYTE_TO_REAL := OutVarREAL;

END_FUNCTION

// ---- Utilities/Helpers/F_GetAdsPort.TcPOU
/// returns the ADS port number used by the current task
FUNCTION F_GetAdsPort : UINT
VAR
	/// FB to get the index of the current task 
	fbTaskIndex: GETCURTASKINDEX;
END_VAR

fbTaskIndex();
F_GetAdsPort := TwinCAT_SystemInfoVarList._TaskInfo[fbTaskIndex.index].AdsPort;

END_FUNCTION

// ---- Utilities/Helpers/P_FilePath.TcPOU
///Programm für die Verzeichnisverwaltung
PROGRAM P_FilePath
VAR_INPUT
	///	path name	
	sPathName: STRING;
	/// 	file name		
	sFileName: STRING;
	///	flag create folder	
	bCreateDIR: BOOL;
	///	flag remove folder	
	bRemoveDIR: BOOL;
END_VAR
VAR_OUTPUT
	///	folder exists flag	
	bFolderExist: BOOL;
END_VAR
VAR
	bBootFolder: BOOL;
	/// 	folders root path 	
	ePath: E_OpenPath;
	///	create DIR	
	fbCreateDir: FB_CreateDir;
	bCreate_Busy: BOOL;
	bCreate_Error: BOOL;
	iCreate_ErrID: UDINT;
	///	delete DIR	
	fbRemoveDir: FB_RemoveDir;
	bRemove_Busy: BOOL;
	bRemove_Error: BOOL;
	iRemove_ErrID: UDINT;
	///	loop		
	iDIR: INT;
END_VAR

///
/// Programm für die Verzeichnisverwaltung
/// 11.05.2012	www.rmth.at
///
(*
	File access program.
	This program is responsible for creating or deleting files.

	Christian Kalser / www.rmth.at / 05.2010
	
	Version:
		0.0.0.1 - Initial Version
*)
(****************************************************************************************)

(*	run program file path	*)
ePath := SEL( bBootFolder, PATH_GENERIC, PATH_BOOTPATH );

CASE iDIR OF

0:
	IF bCreateDIR THEN
		bFolderExist := FALSE;
		bCreateDIR := FALSE;
		fbCreateDir( bExecute := FALSE );
		iDIR := 10;
	ELSIF bRemoveDIR THEN
		bRemoveDIR := FALSE;
		fbRemoveDir( bExecute := FALSE );
		iDIR := 20;
	ELSE
		fbCreateDir( bExecute := FALSE, bBusy=>bCreate_Busy, bError=>bCreate_Error, nErrId=>iCreate_ErrID );
		fbRemoveDir( bExecute := FALSE, bBusy=>bRemove_Busy, bError=>bRemove_Error, nErrId=>iRemove_ErrID );
	END_IF

(*	CREATE DIR		*)
10:
	fbCreateDir(sNetId:= '',
		sPathName:= sPathName,
		ePath:= ePath,
		bExecute:= TRUE,
		tTimeout:= DEFAULT_ADS_TimeOUT,
		bBusy=>bCreate_Busy, bError=>bCreate_Error, nErrId=>iCreate_ErrID );
		iDIR := 12;

12: 	(*	catch error	*)
	fbCreateDir( bExecute := FALSE, bBusy=>bCreate_Busy, bError=>bCreate_Error, nErrId=>iCreate_ErrID );
	IF NOT fbCreateDir.bBusy THEN
		IF NOT fbCreateDir.bError THEN
			bFolderExist := TRUE;
			iDIR := 0;
		ELSE
			CASE iCreate_ErrID OF
				1804: 	(*	folder allready exist	*)
				bFolderExist := TRUE;
				iDIR := 0;
			ELSE
				bFolderExist := FALSE;
				iDIR := 0;
			END_CASE
		END_IF
	END_IF

(*	REMOVE DIR	*)
20:
	fbRemoveDir(sNetId:= '',
		sPathName:= sPathName,
		ePath:= ePath,
		bExecute:= TRUE,
		tTimeout:= DEFAULT_ADS_TimeOUT,
		bBusy=>bRemove_Busy, bError=>bRemove_Error, nErrId=>iRemove_ErrID );
		iDIR := 22;

22: (*	catch error	*)
	fbRemoveDir( bExecute := FALSE, bBusy=>bRemove_Busy, bError=>bRemove_Error, nErrId=>iRemove_ErrID );
	IF NOT fbRemoveDir.bBusy THEN
		IF NOT fbRemoveDir.bError THEN
			bFolderExist := FALSE;
			iDIR := 0;
		ELSE
			CASE iRemove_ErrID OF
				1804:	(*	folder not found	*)
				bFolderExist := FALSE;
				iDIR := 0;
			ELSE
				;
			END_CASE
		END_IF
	END_IF
END_CASE

END_PROGRAM

// ---- Utilities/List/FB_List.TcPOU
FUNCTION_BLOCK FB_List

VAR CONSTANT
	nMaxListEntry						: INT := 255;
END_VAR

VAR		
	stVisu								: Uc_List;
	astEntries							: ARRAY[0..nMaxListEntry] OF ST_Listentry;
	
	
	ptList								: POINTER TO BYTE;
	nEntries							: INT;
	soEntry								: DINT;
	soList								: DINT;
	
END_VAR

METHOD ChangeEntry : E_OperationResult

VAR_INPUT
	Entry					: INT;
	Name					: STRING;
END_VAR
IF Entry < 0 OR Entry > 254 THEN
	RETURN;
END_IF

astEntries[Entry].sName := Name;

Refresh();
END_METHOD

METHOD Clean : BOOL
VAR
	ni			: INT;
END_VAR
IF ptList <> 0 THEN
	MEMSET(ptList, 0, soList);
END_IF

MEMSET(ADR(astEntries), 0, SIZEOF(astEntries));

stVisu.astEntries :=  astEntries;
END_METHOD

METHOD DefineList : BOOL
VAR_INPUT
	List			: ANY;
	Entries			: INT;
END_VAR

VAR
	ni				: INT;
END_VAR
IF Entries > 250 THEN
	RETURN;
END_IF

ptList := List.pValue;
soList := List.diSize;
soEntry := List.diSize/(Entries+1);
nEntries := Entries;
END_METHOD

METHOD InsertEntry : E_OperationResult

VAR_INPUT
	Entry					: INT;
	Name					: STRING;
END_VAR
IF Entry < 0 OR Entry > 254 THEN
	RETURN;
END_IF

MEMMOVE(ADR(astEntries[Entry+1]), ADR(astEntries[Entry]), (nMaxListEntry-Entry-1)*SIZEOF(ST_Listentry));
astEntries[Entry].sName := Name;
astEntries[Entry].bEnable := TRUE;

IF ptList = 0 THEN
	Refresh();
	RETURN;
END_IF


MEMMOVE((ptList + soEntry*(Entry+1)), (ptList + (soEntry*Entry)), (nEntries-Entry-1)*soEntry);
MEMCPY(ptList+Entry*soEntry, ADR(astEntries[Entry]), SIZEOF(ST_Listentry));


Refresh();
END_METHOD

METHOD Load : BOOL
VAR
	ni				: INT;
END_VAR
IF ptList <> 0 THEN

	FOR ni:= 0 TO nEntries DO
		MEMCPY(ADR(astEntries[ni]), ptList+ni*soEntry, SIZEOF(ST_Listentry));
	END_FOR

END_IF

stVisu.astEntries :=  astEntries;
END_METHOD

METHOD MoveEntry : E_OperationResult

VAR_INPUT
	Entry					: INT;
	ToEntry					: INT;
END_VAR
IF ToEntry < 0 OR ToEntry > 254 THEN
	RETURN;
END_IF

MEMMOVE(ADR(astEntries[255]), ADR(astEntries[ToEntry]), SIZEOF(ST_Listentry));
MEMMOVE(ADR(astEntries[ToEntry]), ADR(astEntries[Entry]), SIZEOF(ST_Listentry));
MEMMOVE(ADR(astEntries[Entry]), ADR(astEntries[255]), SIZEOF(ST_Listentry));

IF ptList = 0 THEN
	Refresh();
	RETURN;
END_IF

MEMMOVE(ptList + soEntry*(255), ptList + soEntry*(ToEntry), soEntry);
MEMMOVE(ptList + soEntry*(ToEntry), ptList + soEntry*(Entry), soEntry);
MEMMOVE(ptList + soEntry*(Entry), ptList + soEntry*(255), soEntry);

Refresh();
END_METHOD

METHOD Refresh : BOOL
VAR
	ni				: INT;
END_VAR
IF ptList <> 0 THEN

	FOR ni:= 0 TO nEntries DO	
		MEMCPY(ptList+ni*soEntry, ADR(astEntries[ni]), SIZEOF(ST_Listentry));
	END_FOR
	
END_IF

stVisu.astEntries :=  astEntries;
END_METHOD

METHOD RemoveEntry : E_OperationResult

VAR_INPUT
	Entry			: INT;
END_VAR
IF Entry < 0 OR Entry > 254 THEN
	RETURN;
END_IF

MEMMOVE(ADR(astEntries[Entry]), ADR(astEntries[Entry+1]), (nMaxListEntry-Entry)*SIZEOF(ST_Listentry));

IF ptList = 0 THEN
	Refresh();
	RETURN;
END_IF

MEMMOVE((ptList + (soEntry*Entry)), (ptList + soEntry*(Entry+1)), (nEntries-Entry)*soEntry);

Refresh();
END_METHOD

METHOD Run : BOOL
VAR_INPUT
END_VAR
Visu();
END_METHOD

PROPERTY Selected : UInt
GET
Selected := stVisu.nSelected;
END_GET
END_PROPERTY

PROPERTY SelectedEntry : ST_Listentry
GET
SelectedEntry := astEntries[stVisu.nSelected];
END_GET
END_PROPERTY

PROPERTY SelectedPointer : Pointer TO Byte
GET
SelectedPointer := ptList + (Selected*soEntry);
END_GET
END_PROPERTY

METHOD Visu : BOOL
VAR_INPUT
END_VAR
IF stVisu.bRemove THEN
	stVisu.bRemove := FALSE;
	RemoveEntry(stVisu.nSelected);
	stVisu.astEntries :=  astEntries;
END_IF

IF stVisu.bInsert THEN
	stVisu.bInsert := FALSE;
	InsertEntry(stVisu.nSelected, 'neuer Eintrag');
	stVisu.astEntries :=  astEntries;
END_IF

IF stVisu.bSave THEN
	stVisu.bSave := FALSE;
	astEntries := stVisu.astEntries;
END_IF

IF stVisu.bMoveDown THEN
	stVisu.bMoveDown := FALSE;	
	MoveEntry(stVisu.nSelected, stVisu.nSelected+1);
	stVisu.nSelected := stVisu.nSelected+1;
	stVisu.astEntries :=  astEntries;
END_IF

IF stVisu.bMoveUp THEN
	stVisu.bMoveUp := FALSE;	
	MoveEntry(stVisu.nSelected, stVisu.nSelected-1);
	stVisu.nSelected := stVisu.nSelected-1;
	stVisu.astEntries :=  astEntries;
END_IF

stVisu.ptSelected := SelectedPointer;
END_METHOD

END_FUNCTION_BLOCK

// ---- GlobalTextList.TcGTLO
TEXTLIST GlobalTextList
  646 = '%s'
  993 = '%s Errors'
  1741 = '%s Messages'
  1112 = '%s Warnings'
  1298 = '+'
  394 = '-'
  3091 = 'Clear'
  3875 = 'Mute'
  5707 = '▲'
  2130 = '▼'
  1783 = '⚠'
END_TEXTLIST

// ---- Utilities/List/Visu/Uc_EntryDetail.TcVIS
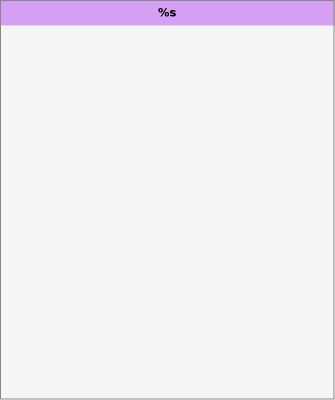
VISUALIZATION Uc_EntryDetail  // 335x400
    Rectangle (0,0 335x25), "%s", text variable: stVisu.sName
        OnMouseClick: write the text variable via Default
    Rectangle (0,26 335x373), text variable: stVisu.sName, colour variable: colCompBg
END_VISUALIZATION
